(* CODESYS project tc3_hbi_mc2.library
   Company: BeckHoff
   DefaultNamespace: Tc3_HBI_MC2
   Version: 3.7.2.1
   Placeholder: Tc3_HBI_MC2
   Title: Tc3_HBI_MC2

Project tree, tasks and I/O mapping:
  libraries: Tc2_Drive, * (Beckhoff Automation GmbH); Tc2_EtherCAT, * (Beckhoff Automation GmbH); Tc2_MC2, * (Beckhoff Automation GmbH); Tc2_MC2_Drive, * (Beckhoff Automation GmbH); Tc2_Standard, * (Beckhoff Automation GmbH); Tc2_System, * (Beckhoff Automation GmbH); Tc2_Utilities, * (Beckhoff Automation GmbH); Tc3_HBI_System, * (BeckHoff); Tc3_Interfaces, * (Beckhoff Automation GmbH); Tc3_Module, * (Beckhoff Automation GmbH); Tc3_System, * (Beckhoff Automation GmbH)
  MOTION/
    POUs/
      FBs/
        [Internal]/
          DUTs/
            Basic/
              RegCorrection/
                data type _ST_MC2_RegCorrection_Get
                data type _ST_MC2_RegCorrection_Set
              data type _ST_MC2_AX5000_Status
              data type _ST_MC2_AX8000_Status
              data type _ST_MC2_Basic
              data type _ST_MC2_Basic_Status
              data type _ST_MC2_Dynamic
              data type _ST_MC2_EL70xx_Status
              data type _ST_MC2_EL72xx_Status
              data type _ST_MC2_Param1
              data type _ST_MC2_Param2
              data type _ST_MC2_SUB_Param
            Compact/
              data type _ST_MC2_Compact_Status
        Basic/
          DUTs/
            data type E_MC2_AX5000_Brake
            data type E_MC2_AX8000_Brake
            data type ST_MC2_AX5000
            data type ST_MC2_AX8000
            data type ST_MC2_Basic
            data type ST_MC2_EL70xx
            data type ST_MC2_EL72xx
            data type ST_MC2_RegCorrection
          ITFs/
            interface I_MC2_AX5000: M_nMC_AcceptBlockedDriveSignal, M_nMC_Brake, M_nMC_ClrLagError, M_nMC_MotorParam1, M_nMC_PID_PosCtrl, M_nMC_Power, M_nMC_Torque, M_nMC_TouchProbe1, M_nMC_TouchProbe2, M_nReset, P_lrRecordedPosition1_RisingEdge, P_lrRecordedPosition2_FallingEdge, P_lrRecordedPosition2_RisingEdge, P_nDiagnosticNumber, P_rActualMainVoltage, P_rAmplifierTemperature, P_rMotorTemperature, P_sDiagnosticNumber
            interface I_MC2_Basic: M_nMC_ClrLagError, M_nMC_DeadTimeComp, M_nMC_GearIn, M_nMC_GearInDyn, M_nMC_GearInMultiMaster, M_nMC_GearOut, M_nMC_InverseMotor, M_nMC_PhasingAbsolute, M_nMC_PhasingRelative, M_nMC_PositionLagMonitoring, M_nMC_Power, M_nMC_RegCorrection, M_nMC_SetEncoderOffset, M_nMC_SetFeedConstant, M_nMC_SetModuloFactor, M_nMC_SetPosition, M_nMC_SetPositionRelative, M_nMC_SetScaleFactor, M_nMC_SetVeloKvFactor, M_nReset, P_bAdvancedSlaveDynamics, P_bInGear, P_lrAbsolutePhaseShift, P_lrCoveredPhaseShift, P_lrGearRatio1, P_lrGearRatio2, P_lrGearRatio3, P_lrGearRatio4, P_lrMaxVelocity, P_lrModuloFactor
            interface I_MC2_EL70xx: P_rAmplifierTemperature, P_rControlVoltage, P_rMotorSupplyVoltage
            interface I_MC2_EL72xx: P_rAmplifierTemperature, P_rMotorSupplyVoltage, P_rMotorTemperature
          function block FB_MC2_AX5000 [ST]: M_nMC_AcceptBlockedDriveSignal, M_nMC_Brake, M_nMC_ClrLagError, M_nMC_DriveData, M_nMC_MotorParam1, M_nMC_PID_PosCtrl, M_nMC_Power, M_nMC_Torque, M_nMC_TouchProbe1, M_nMC_TouchProbe2, M_nReset, P_lrRecordedPosition1_RisingEdge, P_lrRecordedPosition2_FallingEdge, P_lrRecordedPosition2_RisingEdge, P_nDiagnosticNumber, P_rActualMainVoltage, P_rAmplifierTemperature, P_rMotorTemperature, P_sDiagnosticNumber
          function block FB_MC2_AX8000 [ST]: M_nMC_Brake, M_nMC_DriveData, M_nMC_Power, M_nMC_Torque, M_nReset, P_rActualMainVoltage, P_rAmplifierTemperature, P_rMotorTemperature
          function block FB_MC2_Basic [ST]: M_nMC_ClrLagError, M_nMC_DeadTimeComp, M_nMC_GearIn, M_nMC_GearInDyn, M_nMC_GearInMultiMaster, M_nMC_GearOut, M_nMC_InverseMotor, M_nMC_PhasingAbsolute, M_nMC_PhasingRelative, M_nMC_PositionLagMonitoring, M_nMC_Power, M_nMC_ReadParameter, M_nMC_RegCorrection, M_nMC_SetEncoderOffset, M_nMC_SetFeedConstant, M_nMC_SetModuloFactor, M_nMC_SetPosition, M_nMC_SetPositionRelative, M_nMC_SetScaleFactor, M_nMC_SetVeloKvFactor, M_nReset, P_bAdvancedSlaveDynamics, P_bInGear, P_lrAbsolutePhaseShift, P_lrCoveredPhaseShift, P_lrGearRatio1, P_lrGearRatio2, P_lrGearRatio3, P_lrGearRatio4, P_lrMaxVelocity, P_lrModuloFactor
          function block FB_MC2_EL70xx [ST]: M_nMC_DriveData, M_nMC_Power, P_rAmplifierTemperature, P_rControlVoltage, P_rMotorSupplyVoltage
          function block FB_MC2_EL72xx [ST]: M_nMC_DriveData, M_nMC_Power, P_rAmplifierTemperature, P_rMotorSupplyVoltage, P_rMotorTemperature
        Compact/
          DUTs/
            data type ST_MC2_Compact
          ITFs/
            interface I_MC2_Compact: M_nMC_Dynamic, M_nMC_Halt, M_nMC_Home, M_nMC_HomeReset, M_nMC_Jog, M_nMC_MoveAbsolute, M_nMC_MoveModulo, M_nMC_MoveRelative, M_nMC_MoveVelocity, M_nMC_Power, M_nMC_QuickStop, M_nMC_Stop, M_nReset, P_bE_Stop, P_bE_StopDelay, P_bEnable, P_bEnable_Negative, P_bEnable_Positive, P_bHardwareConnected, P_bHomed, P_eBufferMode, P_lrOverride, P_pAXIS_REF, P_pDriveAddress, P_stDynamic
          function block FB_MC2_Compact [ST]: M_nMC_Dynamic, M_nMC_Halt, M_nMC_Home, M_nMC_HomeReset, M_nMC_Jog, M_nMC_Local_Halt, M_nMC_MoveAbsolute, M_nMC_MoveModulo, M_nMC_MoveRelative, M_nMC_MoveVelocity, M_nMC_Power, M_nMC_QuickStop, M_nMC_ReadDriveAddress, M_nMC_Stop, M_nReset, P_bE_Stop, P_bE_StopDelay, P_bEnable, P_bEnable_Negative, P_bEnable_Positive, P_bHardwareConnected, P_bHomed, P_eBufferMode, P_lrOverride, P_pAXIS_REF, P_pDriveAddress, P_sMessage, P_stDynamic
          function block FB_MC2_Compact_AX8000 [ST]: M_nMC_DriveData, M_nMC_Power, M_nReset, P_rActualMainVoltage, P_rAmplifierTemperature, P_rMotorTemperature
  Version/
    global variables Global_Version
  Tc3_HBI_MC2.tmc
*)

// MOTION/POUs/FBs/[Internal]/DUTs/Basic/RegCorrection/_ST_MC2_RegCorrection_Get
{attribute 'hide'}
TYPE _ST_MC2_RegCorrection_Get :
STRUCT
	bWarning: BOOL; 
	nWarningId: UDINT; 
	lrActualVelocityDiff: LREAL; 
	lrActualDistance: LREAL; 
	lrActualLength: LREAL; 
	lrActualAcceleration: LREAL; 
	lrActualDeceleration: LREAL;
END_STRUCT
END_TYPE

// MOTION/POUs/FBs/[Internal]/DUTs/Basic/RegCorrection/_ST_MC2_RegCorrection_Set
{attribute 'hide'}
TYPE _ST_MC2_RegCorrection_Set :
STRUCT
	eMode: Tc2_MC2.E_SuperpositionMode:= Tc2_MC2.SUPERPOSITIONMODE_LENGTHREDUCTION_LIMITEDMOTION;
	lrDistance: LREAL:= 10.0; 
	lrVelocityDiff: LREAL:= 30.0; 
	lrAcceleration: LREAL:= 0.0; 
	lrDeceleration: LREAL:= 0.0; 
	lrJerk: LREAL:= 0.0; 
	lrVelocityProcess: LREAL:= 50.0; 
	lrLength: LREAL:= 360.0;
	eOptions: Tc2_MC2.ST_SuperpositionOptions;
END_STRUCT
END_TYPE

// MOTION/POUs/FBs/[Internal]/DUTs/Basic/_ST_MC2_AX5000_Status
TYPE _ST_MC2_AX5000_Status EXTENDS _ST_MC2_Basic_Status:
STRUCT
	nMC_AcceptBlockedDriveSignal: UDINT;	
	nMC_Brake: UDINT;
	nMC_FeedConstant: UDINT;
	nMC_MotorParam1: UDINT;
	nMC_PID_PosCtrl: UDINT;
	nMC_Torque: UDINT;
	nMC_TouchProbe1: UDINT;
	nMC_TouchProbe2: UDINT;
END_STRUCT
END_TYPE

// MOTION/POUs/FBs/[Internal]/DUTs/Basic/_ST_MC2_AX8000_Status
TYPE _ST_MC2_AX8000_Status EXTENDS _ST_MC2_Basic_Status :
STRUCT
	nMC_Brake: UDINT;	
	nMC_Torque: UDINT;
END_STRUCT
END_TYPE

// MOTION/POUs/FBs/[Internal]/DUTs/Basic/_ST_MC2_Basic
TYPE _ST_MC2_Basic EXTENDS Tc3_HBI_System.ST_Basic :
STRUCT
	bEnable: BOOL;
	bEnable_Negative: BOOL;
	bEnable_Positive: BOOL;
	lrOverride: LREAL;
	lrQuickStopRamp: LREAL;
	bE_Stop: BOOL;
	bE_StopDelay: BOOL;
	bExecute: BOOL;	
	bHome: BOOL;
	bResetHomed: BOOL;	
	bCalibrationCam	: BOOL;
	lrHomePosition	: LREAL;
	bHalt	: BOOL;
	bStop	: BOOL;
	bAbsMove	: BOOL;
	lrAbsPosition	: LREAL;
	lrAbsVelocity	: LREAL;
	bRelMove	: BOOL;
	lrRelDistance	: LREAL;
	lrRelVelocity	: LREAL;
	bMoveVelo	: BOOL;
	lrVeloVelocity	: LREAL;
	bJogForward: BOOL;
	bJogBackwards: BOOL;
	lrJogVelocity	: LREAL;
	lrAcceleration	: LREAL;
	lrDecelaration	: LREAL;
	lrJerk			: LREAL;
	bMoveModulo	: BOOL;
	lrModuloPosition	: LREAL;
	lrModuloVelocity	: LREAL;
	bSetDynamic	: BOOL;
	bReadDriveAddress	: BOOL;
	bPositiveLimit	: BOOL;							
	bNegativeLimit	: BOOL;	

	bSetEncoderOffset: BOOL;
	lrEncoderOffset: LREAL;
	bSetPosition: BOOL;
	lrSetPosotion	: LREAL;						
	
	eBufferMode	: Tc2_MC2.MC_BufferMode;
	eHomingMode	: Tc2_MC2.MC_HomingMode;
	eJogMode		: Tc2_MC2.E_JogMode;
	eDirection		: Tc2_MC2.MC_Direction;
	tHomeTimeout	: TIME;
	tMovementTimeout: TIME;

	bInGear: BOOL;
	lrGearRatio1: LREAL;
	lrGearRatio2: LREAL;
	lrGearRatio3: LREAL;
	lrGearRatio4: LREAL;
	lrModuloFactor: LREAL;
	lrMaxVelocity: LREAL;
	lrAbsolutePhaseShift: LREAL;
	lrCoveredPhaseShift: LREAL;
	stRegCorrection_Get: _ST_MC2_RegCorrection_Get;
END_STRUCT
END_TYPE

// MOTION/POUs/FBs/[Internal]/DUTs/Basic/_ST_MC2_Basic_Status
TYPE _ST_MC2_Basic_Status EXTENDS _ST_MC2_Compact_Status:
STRUCT
	nMC_ClrLagError: UDINT;
	nMC_DeadTimeComp: UDINT;
	nMC_GearIn: UDINT;
	nMC_GearInDyn: UDINT;
	nMC_GearInMultiMaster: UDINT;
	nMC_GearInMultiMaster_Dynamic : UDINT;
	nMC_GearOut: UDINT;
	nMC_InverseMotor: UDINT;
	nMC_PositionLagMonitoring: UDINT;
	nMC_RegCorrection: UDINT;
	nMC_SetFeedConstant: UDINT;
	nMC_SetEncoderOffset: UDINT;
	nMC_SetModuloFactor: UDINT;
	nMC_SetVeloKvFactor: UDINT;
	nMC_SetPosition: UDINT;
	nMC_SetPositionRelative: UDINT;
	nMC_SetScaleFactor: UDINT;
	nMC_PhasingAbsolute: UDINT;
	nMC_PhasingRelative: UDINT;
END_STRUCT
END_TYPE

// MOTION/POUs/FBs/[Internal]/DUTs/Basic/_ST_MC2_Dynamic
TYPE _ST_MC2_Dynamic :
STRUCT
	lrAcceleration: LREAL;
	lrDeceleration: LREAL;
	lrJerk: LREAL;
END_STRUCT
END_TYPE

// MOTION/POUs/FBs/[Internal]/DUTs/Basic/_ST_MC2_EL70xx_Status
TYPE _ST_MC2_EL70xx_Status EXTENDS _ST_MC2_Basic_Status:
STRUCT
END_STRUCT
END_TYPE

// MOTION/POUs/FBs/[Internal]/DUTs/Basic/_ST_MC2_EL72xx_Status
TYPE _ST_MC2_EL72xx_Status EXTENDS _ST_MC2_Basic_Status:
STRUCT
END_STRUCT
END_TYPE

// MOTION/POUs/FBs/[Internal]/DUTs/Basic/_ST_MC2_Param1
{attribute 'hide'}
TYPE _ST_MC2_Param1 :
STRUCT
	aParm: ARRAY[1..6] OF _ST_MC2_SUB_Param;
	nEncoderDir: WORD;
	nMotorDir: WORD;
	nHomeCamDir: WORD;
	nHomeSyncDir: WORD;
	lrRefVelocity: LREAL;
	lrMaxVelocity: LREAL;
END_STRUCT
END_TYPE

// MOTION/POUs/FBs/[Internal]/DUTs/Basic/_ST_MC2_Param2
{attribute 'hide'}
TYPE _ST_MC2_Param2 :
STRUCT
	aParm: ARRAY[1..4] OF _ST_MC2_SUB_Param;
	nEncoderDir: WORD;
	nMotorDir: WORD;
	nHomeCamDir: WORD;
	nHomeSyncDir: WORD;
END_STRUCT
END_TYPE

// MOTION/POUs/FBs/[Internal]/DUTs/Basic/_ST_MC2_SUB_Param
{attribute 'hide'}
TYPE _ST_MC2_SUB_Param :
STRUCT
	nIndexGroup: UDINT;
	nIndexOffset: UDINT;
	nDataSize: UDINT;
END_STRUCT
END_TYPE

// MOTION/POUs/FBs/[Internal]/DUTs/Compact/_ST_MC2_Compact_Status
TYPE _ST_MC2_Compact_Status:
STRUCT
	bHomed: BOOL;
	lrActPos: LREAL;
	lrActVelocity: LREAL;
	nMC_Dynamic: UDINT;
	nMC_Halt: UDINT;
	nMC_Home: UDINT;
	nMC_HomeReset: UDINT;
	nMC_Jog: UDINT;
	M_nMC_Local_Halt: UDINT;
	nMC_MoveAbsolute: UDINT;
	nMC_MoveModulo: UDINT;
	nMC_MoveRelative: UDINT;
	nMC_MoveVelocity: UDINT;
	nMC_Power: UDINT;
	nMC_QuickStop: UDINT;
	M_nMC_ReadDriveAddress: UDINT;
	nMC_Stop: UDINT;
	nReset: UDINT;
END_STRUCT
END_TYPE

// MOTION/POUs/FBs/Basic/DUTs/E_MC2_AX5000_Brake
TYPE E_MC2_AX5000_Brake :
(
	AX5000_Brake_Automatic,	
	AX5000_Brake_Force_lock,	
	AX5000_Brake_Force_unlock
);
END_TYPE

// MOTION/POUs/FBs/Basic/DUTs/E_MC2_AX8000_Brake
TYPE E_MC2_AX8000_Brake :
(
	AX8000_Brake_Release_force,	
	AX8000_Brake_Force_lock,	
	AX8000_Brake_Force_unlock
);
END_TYPE

// MOTION/POUs/FBs/Basic/DUTs/ST_MC2_AX5000
TYPE ST_MC2_AX5000 EXTENDS _ST_MC2_Basic :
STRUCT
	lrRecordedPosition1_RisingEdge: LREAL;
	lrRecordedPosition2_RisingEdge: LREAL;	
	lrRecordedPosition2_FallingEdge: LREAL;		
	rActualMainVoltage: REAL;
	rAmplifierTemperature: REAL;
	rMotorTemperature: REAL;
	nDiagnosticNumber: UDINT;
	sDiagnosticNumber: STRING;
	stStatus: _ST_MC2_AX5000_Status;
END_STRUCT
END_TYPE

// MOTION/POUs/FBs/Basic/DUTs/ST_MC2_AX8000
TYPE ST_MC2_AX8000 EXTENDS _ST_MC2_Basic :
STRUCT
	rActualMainVoltage: REAL;
	rAmplifierTemperature: REAL;
	rMotorTemperature: REAL;
	stStatus: _ST_MC2_AX8000_Status;
END_STRUCT
END_TYPE

// MOTION/POUs/FBs/Basic/DUTs/ST_MC2_Basic
TYPE ST_MC2_Basic EXTENDS _ST_MC2_Basic :
STRUCT
	stStatus: _ST_MC2_Basic_Status;
END_STRUCT
END_TYPE

// MOTION/POUs/FBs/Basic/DUTs/ST_MC2_EL70xx
TYPE ST_MC2_EL70xx EXTENDS _ST_MC2_Basic :
STRUCT
	rAmplifierTemperature: REAL;
	rControlVoltage: REAL;
	rMotorSupplyVoltage: REAL;
	stStatus: _ST_MC2_EL70xx_Status;
END_STRUCT
END_TYPE

// MOTION/POUs/FBs/Basic/DUTs/ST_MC2_EL72xx
TYPE ST_MC2_EL72xx EXTENDS _ST_MC2_Basic :
STRUCT
	rAmplifierTemperature: REAL;
	rMotorSupplyVoltage: REAL;
	rMotorTemperature: REAL;
	stStatus: _ST_MC2_EL72xx_Status;
END_STRUCT
END_TYPE

// MOTION/POUs/FBs/Basic/DUTs/ST_MC2_RegCorrection
TYPE ST_MC2_RegCorrection :
STRUCT
	Set: _ST_MC2_RegCorrection_Set;
	Get: _ST_MC2_RegCorrection_Get;  	
END_STRUCT
END_TYPE

// MOTION/POUs/FBs/Compact/DUTs/ST_MC2_Compact
TYPE ST_MC2_Compact EXTENDS ST_Basic :
STRUCT
	bEnable: BOOL;
	bEnable_Negative: BOOL;
	bEnable_Positive: BOOL;
	lrOverride: LREAL;
	lrQuickStopRamp: LREAL;
	bE_Stop: BOOL;
	bE_StopDelay: BOOL;
	bExecute: BOOL;	
	bHome: BOOL;
	bResetHomed: BOOL;	
	bCalibrationCam	: BOOL;
	lrHomePosition	: LREAL;
	bHalt	: BOOL;
	bStop	: BOOL;
	bAbsMove	: BOOL;
	lrAbsPosition	: LREAL;
	lrAbsVelocity	: LREAL;
	bRelMove	: BOOL;
	lrRelDistance	: LREAL;
	lrRelVelocity	: LREAL;
	bMoveVelo	: BOOL;
	lrVeloVelocity	: LREAL;
	bJogForward: BOOL;
	bJogBackwards: BOOL;
	lrJogVelocity	: LREAL;
	lrAcceleration	: LREAL;
	lrDecelaration	: LREAL;
	lrJerk			: LREAL;
	bMoveModulo	: BOOL;
	lrModuloPosition	: LREAL;
	lrModuloVelocity	: LREAL;
	bSetDynamic	: BOOL;
	bReadDriveAddress	: BOOL;
	bPositiveLimit	: BOOL;							
	bNegativeLimit	: BOOL;							
	eBufferMode	: Tc2_MC2.MC_BufferMode;
	eHomingMode	: Tc2_MC2.MC_HomingMode;
	eJogMode		: Tc2_MC2.E_JogMode;
	eDirection		: Tc2_MC2.MC_Direction;
	tHomeTimeout	: TIME;
	tMovementTimeout: TIME;
	stStatus: _ST_MC2_Compact_Status;
END_STRUCT
END_TYPE

// Version/Global_Version
{attribute 'TcGenerated'}
// This function has been automatically generated from the project information.
VAR_GLOBAL CONSTANT
	{attribute 'const_non_replaced'}
	{attribute 'linkalways'}
	stLibVersion_Tc3_HBI_MC2 : ST_LibVersion := (iMajor := 3, iMinor := 7, iBuild := 2, iRevision := 1, sVersion := '3.7.2.1');
END_VAR

// MOTION/POUs/FBs/Basic/ITFs/I_MC2_AX5000
INTERFACE I_MC2_AX5000 EXTENDS I_MC2_Basic

//	The result of the method is an unsigned double integer
//	0 = idle 
//	1 = coupled
//	2 = starting
//	3 = running
//	4 = aborted
// 	5 = no hardware connected
// 	6 = Spare
//	7 = pointer or index error
//	8 = mapping error
//	9 = parameter error
//	10 = complete
//	Any other number = ErrorID
METHOD PUBLIC M_nMC_AcceptBlockedDriveSignal : UDINT
VAR_INPUT
	bExecute: BOOL;
END_VAR
END_METHOD

//	The result of the method is an unsigned double integer
//	0 = idle 
//	1 = coupled
//	2 = starting
//	3 = running
//	4 = aborted
// 	5 = no hardware connected
// 	6 = Spare
//	7 = pointer or index error
//	8 = mapping error
//	9 = parameter error
//	10 = complete
//	Any other number = ErrorID
METHOD PUBLIC M_nMC_Brake : UDINT
VAR_INPUT
	bExecute: BOOL;
	eBrakeState: E_MC2_AX5000_Brake;
END_VAR
END_METHOD

//	The result of the method is an unsigned double integer
//	0 = idle 
//	1 = coupled
//	2 = starting
//	3 = running
//	4 = aborted
// 	5 = no hardware connected
// 	6 = Spare
//	7 = pointer or index error
//	8 = mapping error
//	9 = parameter error
//	10 = complete
//	Any other number = ErrorID
METHOD PUBLIC M_nMC_ClrLagError : UDINT
VAR_INPUT
	bExecute: BOOL;
END_VAR
END_METHOD

//	The result of the method is an unsigned double integer
//	0 = idle 
//	1 = coupled
//	2 = starting
//	3 = running
//	4 = aborted
// 	5 = no hardware connected
// 	6 = Spare
//	7 = pointer or index error
//	8 = mapping error
//	9 = parameter error
//	10 = complete
//	Any other number = ErrorID
METHOD PUBLIC M_nMC_MotorParam1 : UDINT
VAR_INPUT
	bExecute: BOOL;
	bInverse: BOOL;
	nMaxRpm: UINT;
	lrDiameter: LREAL;
	lrGearNumerator: LREAL;
	lrGearDenominator: LREAL;
END_VAR
END_METHOD

//	The result of the method is an unsigned double integer
//	0 = idle 
//	1 = coupled
//	2 = starting
//	3 = running
//	4 = aborted
// 	5 = no hardware connected
// 	6 = Spare
//	7 = pointer or index error
//	8 = mapping error
//	9 = parameter error
//	10 = complete
//	Any other number = ErrorID
METHOD PUBLIC M_nMC_PID_PosCtrl : UDINT
VAR_INPUT
	bExecute: BOOL;
	rKv: REAL; 		// 0.0 - 100.0 
END_VAR
END_METHOD

//	The result of the method is an unsigned double integer
//	0 = idle 
//	1 = coupled
//	2 = starting
//	3 = running
//	4 = aborted
// 	5 = no hardware connected
// 	6 = Spare
//	7 = pointer or index error
//	8 = mapping error
//	9 = parameter error
//	10 = complete
//	Any other number = ErrorID
METHOD PUBLIC M_nMC_Power : UDINT
VAR_INPUT
	bEnable: BOOL;
	bE_Stop: BOOL;
	bE_StopDelay: BOOL;
	bEnable_Positive: BOOL;
	bEnable_Negative: BOOL;
END_VAR
END_METHOD

//	The result of the method is an unsigned double integer
//	0 = idle 
//	1 = coupled
//	2 = starting
//	3 = running
//	4 = aborted
// 	5 = no hardware connected
// 	6 = Spare
//	7 = pointer or index error
//	8 = mapping error
//	9 = parameter error
//	10 = complete
//	Any other number = ErrorID
METHOD PUBLIC M_nMC_Torque : UDINT
VAR_INPUT
	bExecute: BOOL;
	lrTorque: LREAL; 		// Torque limit 0.0-100.0%	
END_VAR
END_METHOD

//	The result of the method is an unsigned double integer
//	0 = idle 
//	1 = coupled
//	2 = starting
//	3 = running
//	4 = aborted
// 	5 = no hardware connected
// 	6 = Spare
//	7 = pointer or index error
//	8 = mapping error
//	9 = parameter error
//	10 = complete
//	Any other number = ErrorID
METHOD PUBLIC M_nMC_TouchProbe1 : UDINT
VAR_INPUT
	bEnable: BOOL;
	lrPrellFilter_RisingEdge: LREAL;
END_VAR
END_METHOD

//	The result of the method is an unsigned double integer
//	0 = idle 
//	1 = coupled
//	2 = starting
//	3 = running
//	4 = aborted
// 	5 = no hardware connected
// 	6 = Spare
//	7 = pointer or index error
//	8 = mapping error
//	9 = parameter error
//	10 = complete
//	Any other number = ErrorID
METHOD PUBLIC M_nMC_TouchProbe2 : UDINT
VAR_INPUT
	bEnable: BOOL;
	lrPrellFilter_RisingEdge: LREAL;
	lrPrellFilter_FallingEdge: LREAL;
END_VAR
END_METHOD

//	The result of the method is an unsigned double integer
//	0 = idle 
//	1 = coupled
//	2 = starting
//	3 = running
//	4 = aborted
// 	5 = no hardware connected
// 	6 = Spare
//	7 = pointer or index error
//	8 = mapping error
//	9 = parameter error
//	10 = complete
//	Any other number = ErrorID
METHOD PUBLIC M_nReset : UDINT
VAR_INPUT
	bExecute: BOOL;
END_VAR
END_METHOD

PROPERTY PUBLIC P_lrRecordedPosition1_RisingEdge : LREAL
GET
END_GET
END_PROPERTY

PROPERTY PUBLIC P_lrRecordedPosition2_FallingEdge : LREAL
GET
END_GET
END_PROPERTY

PROPERTY PUBLIC P_lrRecordedPosition2_RisingEdge : LREAL
GET
END_GET
END_PROPERTY

PROPERTY PUBLIC P_nDiagnosticNumber : UDINT
GET
END_GET
END_PROPERTY

PROPERTY PUBLIC P_rActualMainVoltage : REAL
GET
END_GET
END_PROPERTY

PROPERTY PUBLIC P_rAmplifierTemperature : REAL
GET
END_GET
END_PROPERTY

PROPERTY PUBLIC P_rMotorTemperature : REAL
GET
END_GET
END_PROPERTY

PROPERTY PUBLIC P_sDiagnosticNumber : STRING
GET
END_GET
END_PROPERTY

END_INTERFACE

// MOTION/POUs/FBs/Basic/ITFs/I_MC2_Basic
INTERFACE I_MC2_Basic EXTENDS I_MC2_Compact

//	The result of the method is an unsigned double integer
//	0 = idle 
//	1 = coupled
//	2 = starting
//	3 = running
//	4 = aborted
// 	5 = no hardware connected
// 	6 = Spare
//	7 = pointer or index error
//	8 = mapping error
//	9 = parameter error
//	10 = complete
//	Any other number = ErrorID
METHOD PUBLIC M_nMC_ClrLagError : UDINT
VAR_INPUT
	bExecute: BOOL;
END_VAR
END_METHOD

//	The result of the method is an unsigned double integer
//	0 = idle 
//	1 = coupled
//	2 = starting
//	3 = running
//	4 = aborted
// 	5 = no hardware connected
// 	6 = Spare
//	7 = pointer or index error
//	8 = mapping error
//	9 = parameter error
//	10 = complete
//	Any other number = ErrorID
METHOD PUBLIC M_nMC_DeadTimeComp : UDINT
END_METHOD

//	The result of the method is an unsigned double integer
//	0 = idle 
//	1 = coupled
//	2 = starting
//	3 = running
//	4 = aborted
// 	5 = no hardware connected
// 	6 = Spare
//	7 = pointer or index error
//	8 = mapping error
//	9 = parameter error
//	10 = complete
//	Any other number = ErrorID
METHOD PUBLIC M_nMC_GearIn : UDINT
VAR_INPUT
	bExecute: BOOL;
	pMaster: POINTER TO TC2_MC2.AXIS_REF;
	lrRatioNumerator: LREAL;
	iRatioDenominator: UINT;
END_VAR
END_METHOD

//	The result of the method is an unsigned double integer
//	0 = idle 
//	1 = coupled
//	2 = starting
//	3 = running
//	4 = aborted
// 	5 = no hardware
//	7 = pointer or index error
//	8 = mapping error
//	9 = parameter error
//	10 = complete
//	Any other number = ErrorID
METHOD PUBLIC M_nMC_GearInDyn : UDINT
VAR_INPUT
	bEnable: BOOL;
	pMaster: POINTER TO TC2_MC2.AXIS_REF;
	lrGearRatio: LREAL;
END_VAR
END_METHOD

//	The result of the method is an unsigned double integer
//	0 = idle 
//	1 = coupled
//	2 = starting
//	3 = running
//	4 = aborted
// 	5 = no hardware connected
// 	6 = Spare
//	7 = pointer or index error
//	8 = mapping error
//	9 = parameter error
//	10 = complete
//	Any other number = ErrorID
METHOD PUBLIC M_nMC_GearInMultiMaster : UDINT
VAR_INPUT
	bEnable: BOOL;
	pMaster1: POINTER TO Tc2_MC2.AXIS_REF;
	pMaster2: POINTER TO Tc2_MC2.AXIS_REF;
	pMaster3: POINTER TO Tc2_MC2.AXIS_REF;
	pMaster4: POINTER TO Tc2_MC2.AXIS_REF;
END_VAR
END_METHOD

//	The result of the method is an unsigned double integer
//	0 = idle 
//	1 = coupled
//	2 = starting
//	3 = running
//	4 = aborted
// 	5 = no hardware connected
// 	6 = Spare
//	7 = pointer or index error
//	8 = mapping error
//	9 = parameter error
//	10 = complete
//	Any other number = ErrorID
METHOD PUBLIC M_nMC_GearOut : UDINT
VAR_INPUT
	bExecute: BOOL;
END_VAR
END_METHOD

//	The result of the method is an unsigned double integer
//	0 = idle 
//	1 = coupled
//	2 = starting
//	3 = running
//	4 = aborted
// 	5 = no hardware connected
// 	6 = Spare
//	7 = pointer or index error
//	8 = mapping error
//	9 = parameter error
//	10 = complete
//	Any other number = ErrorID
METHOD PUBLIC M_nMC_InverseMotor : UDINT
VAR_INPUT
	bExecute: BOOL;
	bInverse: BOOL;
END_VAR
END_METHOD

//	The result of the method is an unsigned double integer
//	0 = idle 
//	1 = coupled
//	2 = starting
//	3 = running
//	4 = aborted
// 	5 = no hardware connected
// 	6 = Spare
//	7 = pointer or index error
//	8 = mapping error
//	9 = parameter error
//	10 = complete
//	Any other number = ErrorID
METHOD PUBLIC M_nMC_PhasingAbsolute : UDINT
VAR_INPUT
	bExecute: BOOL;
	pMaster: POINTER TO TC2_MC2.AXIS_REF;
	lrPhaseShift: LREAL;
	lrVelocity: LREAL;
END_VAR
END_METHOD

//	The result of the method is an unsigned double integer
//	0 = idle 
//	1 = coupled
//	2 = starting
//	3 = running
//	4 = aborted
// 	5 = no hardware connected
// 	6 = Spare
//	7 = pointer or index error
//	8 = mapping error
//	9 = parameter error
//	10 = complete
//	Any other number = ErrorID
METHOD PUBLIC M_nMC_PhasingRelative : UDINT
VAR_INPUT
	bExecute: BOOL;
	pMaster: POINTER TO TC2_MC2.AXIS_REF;
	lrPhaseShift: LREAL;
	lrVelocity: LREAL;
END_VAR
END_METHOD

//	The result of the method is an unsigned double integer
//	0 = idle 
//	1 = coupled
//	2 = starting
//	3 = running
//	4 = aborted
// 	5 = no hardware connected
// 	6 = Spare
//	7 = pointer or index error
//	8 = mapping error
//	9 = parameter error
//	10 = complete
//	Any other number = ErrorID
METHOD PUBLIC M_nMC_PositionLagMonitoring : UDINT
VAR_INPUT
	bEnable: BOOL;
	bDisable: BOOL;
END_VAR
END_METHOD

//	The result of the method is an unsigned double integer
//	0 = idle 
//	1 = coupled
//	2 = starting
//	3 = running
//	4 = aborted
// 	5 = no hardware connected
// 	6 = Spare
//	7 = pointer or index error
//	8 = mapping error
//	9 = parameter error
//	10 = complete
//	Any other number = ErrorID
METHOD PUBLIC M_nMC_Power : UDINT
VAR_INPUT
	bEnable: BOOL;
	bE_Stop: BOOL;
	bE_StopDelay: BOOL;
	bEnable_Positive: BOOL;
	bEnable_Negative: BOOL;
END_VAR
END_METHOD

//	The result of the method is an unsigned double integer
//	0 = idle 
//	1 = coupled
//	2 = starting
//	3 = running
//	4 = aborted
// 	5 = no hardware connected
// 	6 = Spare
//	7 = pointer or index error
//	8 = mapping error
//	9 = parameter error
//	10 = complete
//	Any other number = ErrorID
METHOD PUBLIC M_nMC_RegCorrection : UDINT
VAR_INPUT
	bExecute: BOOL;
	pRegCorrection: POINTER TO ST_MC2_RegCorrection;
END_VAR
END_METHOD

//	The result of the method is an unsigned double integer
//	0 = idle 
//	1 = coupled
//	2 = starting
//	3 = running
//	4 = aborted
// 	5 = no hardware connected
// 	6 = Spare
//	7 = pointer or index error
//	8 = mapping error
//	9 = parameter error
//	10 = complete
//	Any other number = ErrorID
METHOD PUBLIC M_nMC_SetEncoderOffset : UDINT
VAR_INPUT
	bExecute: BOOL;
	lrOffset: LREAL;
END_VAR
END_METHOD

//	The result of the method is an unsigned double integer
//	0 = idle 
//	1 = coupled
//	2 = starting
//	3 = running
//	4 = aborted
// 	5 = no hardware connected
// 	6 = Spare
//	7 = pointer or index error
//	8 = mapping error
//	9 = parameter error
//	10 = complete
//	Any other number = ErrorID
METHOD PUBLIC M_nMC_SetFeedConstant : UDINT
VAR_INPUT
	bExecute: BOOL;
	lrFeedConstant: LREAL;
END_VAR
END_METHOD

//	The result of the method is an unsigned double integer
//	0 = idle 
//	1 = coupled
//	2 = starting
//	3 = running
//	4 = aborted
// 	5 = no hardware connected
// 	6 = Spare
//	7 = pointer or index error
//	8 = mapping error
//	9 = parameter error
//	10 = complete
//	Any other number = ErrorID
METHOD PUBLIC M_nMC_SetModuloFactor : UDINT
VAR_INPUT
	bExecute: BOOL;
	lrModuloFactor: LREAL;
END_VAR
END_METHOD

//	The result of the method is an unsigned double integer
//	0 = idle 
//	1 = coupled
//	2 = starting
//	3 = running
//	4 = aborted
// 	5 = no hardware connected
// 	6 = Spare
//	7 = pointer or index error
//	8 = mapping error
//	9 = parameter error
//	10 = complete
//	Any other number = ErrorID
METHOD PUBLIC M_nMC_SetPosition : UDINT
VAR_INPUT
	bExecute: BOOL;
	lrPosition: LREAL;
END_VAR
END_METHOD

//	The result of the method is an unsigned double integer
//	0 = idle 
//	1 = coupled
//	2 = starting
//	3 = running
//	4 = aborted
// 	5 = no hardware connected
// 	6 = Spare
//	7 = pointer or index error
//	8 = mapping error
//	9 = parameter error
//	10 = complete
//	Any other number = ErrorID
METHOD PUBLIC M_nMC_SetPositionRelative : UDINT
VAR_INPUT
	bExecute: BOOL;
	lrPosition: LREAL;
END_VAR
END_METHOD

//	The result of the method is an unsigned double integer
//	0 = idle 
//	1 = coupled
//	2 = starting
//	3 = running
//	4 = aborted
// 	5 = no hardware connected
// 	6 = Spare
//	7 = pointer or index error
//	8 = mapping error
//	9 = parameter error
//	10 = complete
//	Any other number = ErrorID
METHOD PUBLIC M_nMC_SetScaleFactor : UDINT
VAR_INPUT
	bExecute: BOOL;
	lrScaleFactor: LREAL;
END_VAR
END_METHOD

//	The result of the method is an unsigned double integer
//	0 = idle 
//	1 = coupled
//	2 = starting
//	3 = running
//	4 = aborted
// 	5 = no hardware connected
// 	6 = Spare
//	7 = pointer or index error
//	8 = mapping error
//	9 = parameter error
//	10 = complete
//	Any other number = ErrorID
METHOD PUBLIC M_nMC_SetVeloKvFactor : UDINT
VAR_INPUT
	bExecute: BOOL;
	lrKvFactor: LREAL;
END_VAR
END_METHOD

//	The result of the method is an unsigned double integer
//	0 = idle 
//	1 = coupled
//	2 = starting
//	3 = running
//	4 = aborted
// 	5 = no hardware connected
// 	6 = Spare
//	7 = pointer or index error
//	8 = mapping error
//	9 = parameter error
//	10 = complete
//	Any other number = ErrorID
METHOD PUBLIC M_nReset : UDINT
VAR_INPUT
	bExecute: BOOL;
END_VAR
END_METHOD

PROPERTY PUBLIC P_bAdvancedSlaveDynamics : BOOL
SET
END_SET
END_PROPERTY

PROPERTY PUBLIC P_bInGear : BOOL
GET
END_GET
END_PROPERTY

PROPERTY PUBLIC P_lrAbsolutePhaseShift  : lreal
GET
END_GET
END_PROPERTY

PROPERTY PUBLIC P_lrCoveredPhaseShift : lreal
GET
END_GET
END_PROPERTY

PROPERTY PUBLIC P_lrGearRatio1 : LREAL
SET
END_SET
END_PROPERTY

PROPERTY PUBLIC P_lrGearRatio2 : LREAL
SET
END_SET
END_PROPERTY

PROPERTY PUBLIC P_lrGearRatio3 : LREAL
SET
END_SET
END_PROPERTY

PROPERTY PUBLIC P_lrGearRatio4 : LREAL
SET
END_SET
END_PROPERTY

PROPERTY PUBLIC P_lrMaxVelocity : LREAL
GET
END_GET
END_PROPERTY

PROPERTY PUBLIC P_lrModuloFactor : LREAL
GET
END_GET
END_PROPERTY

END_INTERFACE

// MOTION/POUs/FBs/Compact/ITFs/I_MC2_Compact
INTERFACE I_MC2_Compact EXTENDS Tc3_HBI_System.I_Basic

//	The result of the method is an unsigned double integer
//	0 = idle 
//	1 = coupled
//	2 = starting
//	3 = running
//	4 = aborted
// 	5 = no hardware connected
// 	6 = Spare
//	7 = pointer or index error
//	8 = mapping error
//	9 = parameter error
//	10 = complete
//	Any other number = ErrorID
METHOD PUBLIC M_nMC_Dynamic : UDINT
VAR_INPUT
	bExecute: BOOL;
	lrAcceleration: LREAL;
	lrDeceleration: LREAL;
	lrJerk: LREAL;
END_VAR
END_METHOD

//	The result of the method is an unsigned double integer
//	0 = idle 
//	1 = coupled
//	2 = starting
//	3 = running
//	4 = aborted
// 	5 = no hardware connected
// 	6 = Spare
//	7 = pointer or index error
//	8 = mapping error
//	9 = parameter error
//	10 = complete
//	Any other number = ErrorID
METHOD PUBLIC M_nMC_Halt : UDINT
VAR_INPUT
	bExecute: BOOL;
END_VAR
END_METHOD

//	The result of the method is an unsigned double integer
//	0 = idle 
//	1 = coupled
//	2 = starting
//	3 = running
//	4 = aborted
// 	5 = no hardware connected
// 	6 = Spare
//	7 = pointer or index error
//	8 = mapping error
//	9 = parameter error
//	10 = complete
//	Any other number = ErrorID
METHOD PUBLIC M_nMC_Home : UDINT
VAR_INPUT
	bExecute: BOOL;
	lrPosition: LREAL;
	bCalibrationCam: BOOL;
	eHomingMode: MC_HomingMode;
END_VAR
END_METHOD

//	The result of the method is an unsigned double integer
//	0 = idle 
//	1 = coupled
//	2 = starting
//	3 = running
//	4 = aborted
// 	5 = no hardware connected
// 	6 = Spare
//	7 = pointer or index error
//	8 = mapping error
//	9 = parameter error
//	10 = complete
//	Any other number = ErrorID
METHOD PUBLIC M_nMC_HomeReset : UDINT
VAR_INPUT
	bExecute: BOOL;
END_VAR
END_METHOD

//	The result of the method is an unsigned double integer
//	0 = idle 
//	1 = coupled
//	2 = starting
//	3 = running
//	4 = aborted
// 	5 = no hardware connected
// 	6 = Spare
//	7 = pointer or index error
//	8 = mapping error
//	9 = parameter error
//	10 = complete
//	Any other number = ErrorID
METHOD PUBLIC M_nMC_Jog : UDINT
VAR_INPUT
	bForward: BOOL;
	bBackwards: BOOL;
	lrVelocity: LREAL;
END_VAR
END_METHOD

//	The result of the method is an unsigned double integer
//	0 = idle 
//	1 = coupled
//	2 = starting
//	3 = running
//	4 = aborted
// 	5 = no hardware connected
// 	6 = Spare
//	7 = pointer or index error
//	8 = mapping error
//	9 = parameter error
//	10 = complete
//	Any other number = ErrorID
METHOD PUBLIC M_nMC_MoveAbsolute : UDINT
VAR_INPUT
	bExecute: BOOL;
	lrPosition: LREAL;
	lrVelocity: LREAL;
END_VAR
END_METHOD

//	The result of the method is an unsigned double integer
//	0 = idle 
//	1 = coupled
//	2 = starting
//	3 = running
//	4 = aborted
// 	5 = no hardware connected
// 	6 = Spare
//	7 = pointer or index error
//	8 = mapping error
//	9 = parameter error
//	10 = complete
//	Any other number = ErrorID
METHOD PUBLIC M_nMC_MoveModulo : UDINT
VAR_INPUT
	bExecute: BOOL;
	lrPosition: LREAL;
	lrVelocity: LREAL;
	eDirection: Tc2_MC2.MC_Direction;
END_VAR
END_METHOD

//	The result of the method is an unsigned double integer
//	0 = idle 
//	1 = coupled
//	2 = starting
//	3 = running
//	4 = aborted
// 	5 = no hardware connected
// 	6 = Spare
//	7 = pointer or index error
//	8 = mapping error
//	9 = parameter error
//	10 = complete
//	Any other number = ErrorID
METHOD PUBLIC M_nMC_MoveRelative : UDINT
VAR_INPUT
	bExecute: BOOL;
	lrDistance: LREAL;
	lrVelocity: LREAL;
END_VAR
END_METHOD

//	The result of the method is an unsigned double integer
//	0 = idle 
//	1 = coupled
//	2 = starting
//	3 = running
//	4 = aborted
// 	5 = no hardware connected
// 	6 = Spare
//	7 = pointer or index error
//	8 = mapping error
//	9 = parameter error
//	10 = complete
//	Any other number = ErrorID
METHOD PUBLIC M_nMC_MoveVelocity : UDINT
VAR_INPUT
	bExecute: BOOL;
	lrVelocity: LREAL;
	eDirection: MC_Direction;
END_VAR
END_METHOD

//	The result of the method is an unsigned double integer
//	0 = idle 
//	1 = coupled
//	2 = starting
//	3 = running
//	4 = aborted
// 	5 = no hardware connected
// 	6 = Spare
//	7 = pointer or index error
//	8 = mapping error
//	9 = parameter error
//	10 = complete
//	Any other number = ErrorID
METHOD PUBLIC M_nMC_Power : UDINT
VAR_INPUT
	bEnable: BOOL;
	bE_Stop: BOOL;
	bE_StopDelay: BOOL;
	bEnable_Positive: BOOL;
	bEnable_Negative: BOOL;
END_VAR
END_METHOD

//	The result of the method is an unsigned double integer
//	0 = idle 
//	1 = coupled
//	2 = starting
//	3 = running
//	4 = aborted
// 	5 = no hardware connected
// 	6 = Spare
//	7 = pointer or index error
//	8 = mapping error
//	9 = parameter error
//	10 = complete
//	Any other number = ErrorID
METHOD PUBLIC M_nMC_QuickStop : UDINT
VAR_INPUT
	bExecute: BOOL;
	lrDeceleration: LREAL;
	lrJerk: LREAL;
END_VAR
END_METHOD

//	The result of the method is an unsigned double integer
//	0 = idle 
//	1 = coupled
//	2 = starting
//	3 = running
//	4 = aborted
// 	5 = no hardware connected
// 	6 = Spare
//	7 = pointer or index error
//	8 = mapping error
//	9 = parameter error
//	10 = complete
//	Any other number = ErrorID
METHOD PUBLIC M_nMC_Stop : UDINT
VAR_INPUT
	bExecute: BOOL;
END_VAR
END_METHOD

//	The result of the method is an unsigned double integer
//	0 = idle 
//	1 = coupled
//	2 = starting
//	3 = running
//	4 = aborted
// 	5 = no hardware connected
// 	6 = Spare
//	7 = pointer or index error
//	8 = mapping error
//	9 = parameter error
//	10 = complete
//	Any other number = ErrorID
METHOD PUBLIC M_nReset : UDINT
VAR_INPUT
	bExecute: BOOL;
END_VAR
END_METHOD

PROPERTY PUBLIC P_bE_Stop : BOOL
GET
END_GET
END_PROPERTY

PROPERTY PUBLIC P_bE_StopDelay : BOOL
GET
END_GET
END_PROPERTY

PROPERTY PUBLIC P_bEnable : BOOL
GET
END_GET
END_PROPERTY

PROPERTY PUBLIC P_bEnable_Negative : BOOL
GET
END_GET
END_PROPERTY

PROPERTY PUBLIC P_bEnable_Positive : BOOL
GET
END_GET
END_PROPERTY

PROPERTY PUBLIC P_bHardwareConnected : BOOL
GET
END_GET
END_PROPERTY

PROPERTY PUBLIC P_bHomed : BOOL
GET
END_GET
END_PROPERTY

PROPERTY PUBLIC P_eBufferMode : MC_BufferMode
SET
END_SET
END_PROPERTY

PROPERTY PUBLIC P_lrOverride : LREAL
GET
END_GET
SET
END_SET
END_PROPERTY

PROPERTY PUBLIC P_pAXIS_REF : POINTER TO AXIS_REF
GET
END_GET
END_PROPERTY

PROPERTY PUBLIC P_pDriveAddress : POINTER TO ST_AdsAddress
GET
END_GET
END_PROPERTY

PROPERTY PUBLIC P_stDynamic : _ST_MC2_Dynamic
GET
END_GET
END_PROPERTY

END_INTERFACE

// MOTION/POUs/FBs/Basic/ITFs/I_MC2_EL70xx
INTERFACE I_MC2_EL70xx EXTENDS I_MC2_Basic

PROPERTY PUBLIC P_rAmplifierTemperature : REAL
GET
END_GET
END_PROPERTY

PROPERTY PUBLIC P_rControlVoltage : REAL
GET
END_GET
END_PROPERTY

PROPERTY PUBLIC P_rMotorSupplyVoltage : REAL
GET
END_GET
END_PROPERTY

END_INTERFACE

// MOTION/POUs/FBs/Basic/ITFs/I_MC2_EL72xx
INTERFACE I_MC2_EL72xx EXTENDS I_MC2_Basic

PROPERTY PUBLIC P_rAmplifierTemperature : REAL
GET
END_GET
END_PROPERTY

PROPERTY PUBLIC P_rMotorSupplyVoltage : REAL
GET
END_GET
END_PROPERTY

PROPERTY PUBLIC P_rMotorTemperature : REAL
GET
END_GET
END_PROPERTY

END_INTERFACE

// MOTION/POUs/FBs/Basic/FB_MC2_AX5000
//------------------------------------------------------------------------------------------
//                                                                                        	
//***************************** Beckhoff TwinCAT Examples **********************************
//                                                                                        	
//************************************* WARNING ********************************************
// This program is only an example. If it is used as a control program in any real        	
// application, Beckhoff is not responsible for any malfunction, loss or damage           	
// which could arise by using this program!                                               	
//                                                                                        	
//*************************************  Program Info. *************************************
//                                                                                        	
// PLC program name:    	FB_MC2_AX5000 (FB)               	                           	
// Hardware platform:      	TwinCat PTP v3.1.4022				                          		                                  	
//                                                                                        	
// ======================================================================================== 
//         Version       Date                        Remarks                              	
// ======================================================================================== 
//         3.1           27 feb 2018                 First release of this example        	
// ======================================================================================== 
//                                                                                        	
//******************************* Aims OF this PLC PROGRAM *********************************
//                                                                                        	 
//                                                                                        	
//----------------------------------------------------------------------------------------- 
FUNCTION_BLOCK FB_MC2_AX5000 EXTENDS FB_MC2_Basic IMPLEMENTS I_MC2_AX5000
VAR
	FB_MC2_AX5000_M_nMC_Brake_bExecute: BOOL;
	FB_MC2_AX5000_M_nMC_Brake_eBrakeState: E_MC2_AX5000_Brake;
	FB_MC2_AX5000_M_nMC_Brake_iState: INT;
	FB_MC2_AX5000_M_nMC_Brake_nValue: UINT;
	FB_MC2_AX5000_M_nMC_Brake_fbExecute_R_TRIG: Tc2_Standard.R_TRIG;
	FB_MC2_AX5000_M_nMC_Brake_fbSoEWrite: TC2_MC2_DRIVE.FB_SoEWrite;

	FB_MC2_AX5000_M_nMC_ClrLagError_bExecute: BOOL;
	FB_MC2_AX5000_M_nMC_ClrLagError_iState: INT;
	FB_MC2_AX5000_M_nMC_ClrLagError_fbExecute_R_TRIG: Tc2_Standard.R_TRIG;
	FB_MC2_AX5000_M_nMC_ClrLagError_fbSoEWrite: TC2_MC2_DRIVE.FB_SoEWrite;
	FB_MC2_AX5000_M_nMC_ClrLagError_nData: UDINT;
	FB_MC2_AX5000_M_nMC_ClrLagError_bDone: BOOL;
	FB_MC2_AX5000_M_nMC_ClrLagError_nStatus: UDINT;

	FB_MC2_AX5000_M_nMC_DriveData_iState: INT;
	FB_MC2_AX5000_M_nMC_DriveData_fbSoEAX5000ReadActMainVoltage: FB_SoEAX5000ReadActMainVoltage;
	FB_MC2_AX5000_M_nMC_DriveData_fbSoEReadAmplifierTemperature: FB_SoEReadAmplifierTemperature;
	FB_MC2_AX5000_M_nMC_DriveData_fbSoEReadMotorTemperature: FB_SoEReadMotorTemperature;
	FB_MC2_AX5000_M_nMC_DriveData_fbSoERead: Tc2_MC2_Drive.FB_SoERead;
	FB_MC2_AX5000_M_nMC_DriveData_lrActualMainVoltage: LREAL;
	FB_MC2_AX5000_M_nMC_DriveData_lrAmplifierTemperature: LREAL;
	FB_MC2_AX5000_M_nMC_DriveData_lrMotorTemperature: LREAL;
	FB_MC2_AX5000_M_nMC_DriveData_nDiagnosticNumber: UDINT;

	FB_MC2_AX5000_M_nMC_MotorParam1_bExecute: BOOL;
	FB_MC2_AX5000_M_nMC_MotorParam1_bInverse: BOOL;
	FB_MC2_AX5000_M_nMC_MotorParam1_nMaxRpm: UINT;
	FB_MC2_AX5000_M_nMC_MotorParam1_lrDiameter: LREAL;
	FB_MC2_AX5000_M_nMC_MotorParam1_lrGearNumerator: LREAL;
	FB_MC2_AX5000_M_nMC_MotorParam1_lrGearDenominator: LREAL;
	FB_MC2_AX5000_M_nMC_MotorParam1_iState: INT;
	FB_MC2_AX5000_M_nMC_MotorParam1_fbExecute_R_TRIG: R_TRIG;
	FB_MC2_AX5000_M_nMC_MotorParam1_fbADSRDWRT: ADSRDWRT;
	FB_MC2_AX5000_M_nMC_MotorParam1_fbMC2_SetEncoderScalingFactor: MC_SetEncoderScalingFactor;
	FB_MC2_AX5000_M_nMC_MotorParam1_stMC2_Param: _ST_MC2_Param1;
	FB_MC2_AX5000_M_nMC_MotorParam1_arr_nADSReturn: ARRAY[1..6] OF UDINT;
	
	FB_MC2_AX5000_M_nMC_PID_PosCtrl_bExecute: BOOL;
	FB_MC2_AX5000_M_nMC_PID_PosCtrl_rKv: REAL; 
	FB_MC2_AX5000_M_nMC_PID_PosCtrl_iState: INT;
	FB_MC2_AX5000_M_nMC_PID_PosCtrl_iKv: INT;
	FB_MC2_AX5000_M_nMC_PID_PosCtrl_fbExecute_R_TRIG: R_TRIG;
	FB_MC2_AX5000_M_nMC_PID_PosCtrl_fbSoEWrite: TC2_MC2_DRIVE.FB_SoEWrite;

	FB_MC2_AX5000_M_nMC_Power_bEnable: BOOL;
	FB_MC2_AX5000_M_nMC_Power_bE_Stop: BOOL;
	FB_MC2_AX5000_M_nMC_Power_bE_StopDelay: BOOL;
	FB_MC2_AX5000_M_nMC_Power_bEnable_Positive: BOOL;
	FB_MC2_AX5000_M_nMC_Power_bEnable_Negative: BOOL;
	FB_MC2_AX5000_M_nMC_Power_fbStartDelay_TON: Tc2_Standard.TON;
	FB_MC2_AX5000_M_nMC_Power_arr_nRet: ARRAY[1..4] OF UDINT;
	
	FB_MC2_AX5000_M_nMC_Torque_bExecute: BOOL;
	FB_MC2_AX5000_M_nMC_Torque_lrTorque: LREAL; 		// Torque limit 0.0-100.0%	
	FB_MC2_AX5000_M_nMC_Torque_iState: INT;
	FB_MC2_AX5000_M_nMC_Torque_iTorque: INT;
	FB_MC2_AX5000_M_nMC_Torque_fbExecute_R_TRIG: R_TRIG;
	FB_MC2_AX5000_M_nMC_Torque_fbSoEWrite: TC2_MC2_DRIVE.FB_SoEWrite;
	
	FB_MC2_AX5000_M_nMC_TouchProbe1_bEnable: BOOL;
	FB_MC2_AX5000_M_nMC_TouchProbe1_lrPrellFilter_RisingEdge: LREAL;
	FB_MC2_AX5000_M_nMC_TouchProbe1_iState: INT;
	FB_MC2_AX5000_M_nMC_TouchProbe1_fbEnable_R_TRIG: R_TRIG;
	FB_MC2_AX5000_M_nMC_TouchProbe1_fbDisable_R_TRIG: R_TRIG;	
	FB_MC2_AX5000_M_nMC_TouchProbe1_fbTouchProbe: Tc2_MC2.MC_TouchProbe;
	FB_MC2_AX5000_M_nMC_TouchProbe1_fbAbortTrigger: Tc2_MC2.MC_AbortTrigger;
	FB_MC2_AX5000_M_nMC_TouchProbe1_stTriggerInput: Tc2_MC2.TRIGGER_REF;
	FB_MC2_AX5000_M_nMC_TouchProbe1_lrRecordedPosition1_RisingEdge: LREAL;
	FB_MC2_AX5000_M_nMC_TouchProbe1_lrLastLatchPosition: LREAL;

	FB_MC2_AX5000_M_nMC_TouchProbe2_bEnable: BOOL;
	FB_MC2_AX5000_M_nMC_TouchProbe2_bRisingEdgeDone: BOOL;
	FB_MC2_AX5000_M_nMC_TouchProbe2_iState: INT;
	FB_MC2_AX5000_M_nMC_TouchProbe2_lrPrellFilter_RisingEdge: LREAL;
	FB_MC2_AX5000_M_nMC_TouchProbe2_lrPrellFilter_FallingEdge: LREAL;
	FB_MC2_AX5000_M_nMC_TouchProbe2_fbEnable_R_TRIG: Tc2_Standard.R_TRIG;
	FB_MC2_AX5000_M_nMC_TouchProbe2_fbDisable_R_TRIG: Tc2_Standard.R_TRIG;	
	FB_MC2_AX5000_M_nMC_TouchProbe2_fbTouchProbe: Tc2_MC2.MC_TouchProbe;
	FB_MC2_AX5000_M_nMC_TouchProbe2_stTriggerInput: Tc2_MC2.TRIGGER_REF;
	FB_MC2_AX5000_M_nMC_TouchProbe2_fbAbortTrigger: Tc2_MC2.MC_AbortTrigger;
	FB_MC2_AX5000_M_nMC_TouchProbe2_lrRecordedPosition2_RisingEdge: LREAL;
	FB_MC2_AX5000_M_nMC_TouchProbe2_lrRecordedPosition2_FallingEdge: LREAL;
	FB_MC2_AX5000_M_nMC_TouchProbe2_lrLastLatchPosition: LREAL;
	
	FB_MC2_AX5000_M_nReset_iState: INT;
	FB_MC2_AX5000_M_nReset_fbExecute_R_TRIG: Tc2_Standard.R_TRIG;
	FB_MC2_AX5000_M_nReset_fbSoEReset: Tc2_MC2_Drive.FB_SoEReset;
	FB_MC2_AX5000_M_nReset_nStatus: UDINT;
END_VAR

//	The result of the method is an unsigned double integer
//	0 = idle 
//	1 = coupled
//	2 = starting
//	3 = running
//	4 = aborted
// 	5 = no hardware connected
// 	6 = Spare
//	7 = pointer or index error
//	8 = mapping error
//	9 = parameter error
//	10 = complete
//	Any other number = ErrorID
METHOD PUBLIC M_nMC_AcceptBlockedDriveSignal : UDINT
VAR_INPUT
	bExecute: BOOL;
END_VAR
// No hardware connected
IF NOT _bHardwareConnected THEN
	Tc2_MC2.MC_SetAcceptBlockedDriveSignal(Axis:= _stAXIS_REF, Enable:= FALSE);
	IF bExecute THEN
		M_nMC_AcceptBlockedDriveSignal:= Tc3_HBI_System.cNO_HARDWARE_CONNECTED;
	END_IF	
	RETURN;
END_IF

// Update function
IF _stAXIS_REF.NcToPlc.AxisID > 0 THEN
	IF _bHardwareConnected THEN
		IF Tc2_MC2.MC_SetAcceptBlockedDriveSignal(Axis:= _stAXIS_REF, Enable:= bExecute) THEN
			M_nMC_AcceptBlockedDriveSignal:= Tc3_HBI_System.cCOMPLETE;
		ELSE
			M_nMC_AcceptBlockedDriveSignal:= Tc3_HBI_System.cIDLE;
		END_IF	
	ELSE
		Tc2_MC2.MC_SetAcceptBlockedDriveSignal(Axis:= _stAXIS_REF, Enable:= FALSE);
		M_nMC_AcceptBlockedDriveSignal:= Tc3_HBI_System.cNO_HARDWARE_CONNECTED;
	END_IF
ELSE
	Tc2_MC2.MC_SetAcceptBlockedDriveSignal(Axis:= _stAXIS_REF, Enable:= FALSE); 
	IF bExecute THEN
		M_nMC_AcceptBlockedDriveSignal:= Tc3_HBI_System.cMAPPING_ERROR;		
	END_IF
	RETURN;
END_IF
END_METHOD

//	The result of the method is an unsigned double integer
//	0 = idle 
//	1 = coupled
//	2 = starting
//	3 = running
//	4 = aborted
// 	5 = no hardware connected
// 	6 = Spare
//	7 = pointer or index error
//	8 = mapping error
//	9 = parameter error
//	10 = complete
//	Any other number = ErrorID
METHOD PUBLIC M_nMC_Brake : UDINT
VAR_INPUT
	bExecute: BOOL;
	eBrakeState: E_MC2_AX5000_Brake;
END_VAR
// Local variable
FB_MC2_AX5000_M_nMC_Brake_bExecute:= bExecute;
FB_MC2_AX5000_M_nMC_Brake_eBrakeState:= eBrakeState;

//**********************************
// Reset 
//**********************************
IF _bReset THEN
	IF _bError THEN
		FB_MC2_AX5000_M_nMC_Brake_fbSoEWrite(Execute:= FALSE, Axis:= _stAXIS_REF); 
		FB_MC2_AX5000_M_nMC_Brake_iState:= 000;
	END_IF
END_IF

// No hardware connected
IF NOT _bHardwareConnected THEN
	FB_MC2_AX5000_M_nMC_Brake_fbSoEWrite(Execute:= FALSE, Axis:= _stAXIS_REF); 
	FB_MC2_AX5000_M_nMC_Brake_iState:= 000;
	IF FB_MC2_AX5000_M_nMC_Brake_bExecute THEN
		M_nMC_Brake:= Tc3_HBI_System.cNO_HARDWARE_CONNECTED;
	END_IF	
	RETURN;
END_IF

// Parameter check 
IF FB_MC2_AX5000_M_nMC_Brake_bExecute THEN
	IF FB_MC2_AX5000_M_nMC_Brake_eBrakeState = AX5000_Brake_Automatic OR FB_MC2_AX5000_M_nMC_Brake_eBrakeState = AX5000_Brake_Force_lock OR FB_MC2_AX5000_M_nMC_Brake_eBrakeState = AX5000_Brake_Force_unlock THEN
		;
	ELSE
		// Parameter error	
		M_nMC_Brake:= Tc3_HBI_System.cPARAMETER_ERROR;
		RETURN;
	END_IF
END_IF

//**********************************
// Wait for execute
//**********************************
IF _stAXIS_REF.NcToPlc.AxisID > 0 THEN
	FB_MC2_AX5000_M_nMC_Brake_fbExecute_R_TRIG(CLK:= FB_MC2_AX5000_M_nMC_Brake_bExecute);
	IF FB_MC2_AX5000_M_nMC_Brake_fbExecute_R_TRIG.Q THEN
		FB_MC2_AX5000_M_nMC_Brake_fbSoEWrite(Execute:= FALSE, Axis:= _stAXIS_REF); 
		FB_MC2_AX5000_M_nMC_Brake_iState:= 001;
	END_IF
ELSE
	FB_MC2_AX5000_M_nMC_Brake_fbSoEWrite(Execute:= FALSE, Axis:= _stAXIS_REF); 
	FB_MC2_AX5000_M_nMC_Brake_iState:= 000;
	IF FB_MC2_AX5000_M_nMC_Brake_bExecute THEN
		M_nMC_Brake:= Tc3_HBI_System.cMAPPING_ERROR;		
	END_IF
	RETURN;
END_IF


//**********************************
// Main sequence
//**********************************
CASE FB_MC2_AX5000_M_nMC_Brake_iState OF

	000: 	// Do nothing
	
	001:	// Set brake state
			M_nMC_Brake:= Tc3_HBI_System.cRUNNING;

			CASE FB_MC2_AX5000_M_nMC_Brake_eBrakeState OF
				
				AX5000_Brake_Automatic:
					FB_MC2_AX5000_M_nMC_Brake_nValue:= 0;

				AX5000_Brake_Force_lock:
					FB_MC2_AX5000_M_nMC_Brake_nValue:= 1;
			
				AX5000_Brake_Force_unlock:
					FB_MC2_AX5000_M_nMC_Brake_nValue:= 2;
				
			ELSE	
				FB_MC2_AX5000_M_nMC_Brake_nValue:= 0;
			END_CASE

			FB_MC2_AX5000_M_nMC_Brake_iState:= FB_MC2_AX5000_M_nMC_Brake_iState +1;

	002:	// Write brake state to AX5000
			M_nMC_Brake:= Tc3_HBI_System.cRUNNING;
			FB_MC2_AX5000_M_nMC_Brake_fbSoEWrite(Execute:= FALSE, Axis:= _stAXIS_REF); 
			FB_MC2_AX5000_M_nMC_Brake_fbSoEWrite(
				NetId:= '', 
				Idn:= P_0_IDN + 96, 
				Element:= 16#40, 
				pSrcBuf:= ADR(FB_MC2_AX5000_M_nMC_Brake_nValue), 
				BufLen:= SIZEOF(FB_MC2_AX5000_M_nMC_Brake_nValue), 
				Execute:= TRUE, 
				Timeout:= Tc2_System.DEFAULT_ADS_TIMEOUT, 
				Password:= , 
				Axis:= _stAXIS_REF, 
				Busy=> , 
				Error=> , 
				AdsErrId=> , 
				SercosErrId=> );
	
			FB_MC2_AX5000_M_nMC_Brake_iState:= FB_MC2_AX5000_M_nMC_Brake_iState +1;

	003:	// Write brake state
			M_nMC_Brake:= Tc3_HBI_System.cRUNNING;
			FB_MC2_AX5000_M_nMC_Brake_fbSoEWrite(Execute:= TRUE, Axis:= _stAXIS_REF); 
			
			// Error handling
			IF FB_MC2_AX5000_M_nMC_Brake_fbSoEWrite.Error THEN
				M_nError(FB_MC2_AX5000_M_nMC_Brake_fbSoEWrite.AdsErrId);
				M_nMC_Brake:= FB_MC2_AX5000_M_nMC_Brake_fbSoEWrite.AdsErrId;
			ELSE
				// Done
				IF NOT FB_MC2_AX5000_M_nMC_Brake_fbSoEWrite.Busy THEN
					FB_MC2_AX5000_M_nMC_Brake_fbSoEWrite(Execute:= FALSE, Axis:= _stAXIS_REF); 
					FB_MC2_AX5000_M_nMC_Brake_iState:= FB_MC2_AX5000_M_nMC_Brake_iState +1;
				END_IF	
			END_IF
		
	004:	// Done
			M_nMC_Brake:= Tc3_HBI_System.cCOMPLETE;
			IF NOT FB_MC2_AX5000_M_nMC_Brake_bExecute THEN
				FB_MC2_AX5000_M_nMC_Brake_iState:= 000;
			END_IF
			
ELSE
	FB_MC2_AX5000_M_nMC_Brake_iState:= 000;
END_CASE
END_METHOD

//	The result of the method is an unsigned double integer
//	0 = idle 
//	1 = coupled
//	2 = starting
//	3 = running
//	4 = aborted
// 	5 = no hardware connected
// 	6 = Spare
//	7 = pointer or index error
//	8 = mapping error
//	9 = parameter error
//	10 = complete
//	Any other number = ErrorID
METHOD PUBLIC M_nMC_ClrLagError : UDINT
VAR_INPUT
	bExecute: BOOL;
END_VAR
// Local varisble
FB_MC2_AX5000_M_nMC_ClrLagError_bExecute:= bExecute;

//**********************************
// Reset 
//**********************************
IF _bReset THEN
	IF _bError THEN
		FB_MC2_AX5000_M_nMC_ClrLagError_fbSoEWrite(Execute:= FALSE, Axis:= _stAXIS_REF); 
		SUPER^.M_nMC_ClrLagError(bExecute:= FALSE);
		FB_MC2_AX5000_M_nMC_ClrLagError_fbExecute_R_TRIG(CLK:= FALSE);
		FB_MC2_AX5000_M_nMC_ClrLagError_iState:= 000;
	END_IF
END_IF
// No hardware connected
IF NOT _bHardwareConnected THEN
	SUPER^.M_nMC_ClrLagError(bExecute:= FALSE);
	FB_MC2_AX5000_M_nMC_ClrLagError_fbExecute_R_TRIG(CLK:= FALSE);
	FB_MC2_AX5000_M_nMC_ClrLagError_iState:= 000;
	IF FB_MC2_AX5000_M_nMC_ClrLagError_bExecute THEN
		M_nMC_ClrLagError:= Tc3_HBI_System.cNO_HARDWARE_CONNECTED;
	END_IF	
	RETURN;
END_IF


//**********************************
// Wait for execute
//**********************************
IF _stAXIS_REF.NcToPlc.AxisID > 0 THEN
	FB_MC2_AX5000_M_nMC_ClrLagError_fbExecute_R_TRIG(CLK:= FB_MC2_AX5000_M_nMC_ClrLagError_bExecute);
	IF FB_MC2_AX5000_M_nMC_ClrLagError_fbExecute_R_TRIG.Q THEN
		FB_MC2_AX5000_M_nMC_ClrLagError_fbSoEWrite(Execute:= FALSE, Axis:= _stAXIS_REF); 
		SUPER^.M_nMC_ClrLagError(bExecute:= FALSE);
		IF FB_MC2_AX5000_M_nMC_ClrLagError_bDone THEN
			FB_MC2_AX5000_M_nMC_ClrLagError_iState:= 010;
		ELSE
			FB_MC2_AX5000_M_nMC_ClrLagError_iState:= 001;
		END_IF
	END_IF
ELSE
	FB_MC2_AX5000_M_nMC_ClrLagError_fbExecute_R_TRIG(CLK:= FALSE);
	FB_MC2_AX5000_M_nMC_ClrLagError_iState:= 000;
	IF FB_MC2_AX5000_M_nMC_ClrLagError_bExecute THEN
		M_nMC_ClrLagError:= Tc3_HBI_System.cMAPPING_ERROR;
	END_IF
	RETURN;
END_IF


//**********************************
// Main sequence
//**********************************
CASE FB_MC2_AX5000_M_nMC_ClrLagError_iState OF

	000: 	// Do nothing
	
	001:	// Reset lag error S_0_159 = 0	
			M_nMC_ClrLagError:= Tc3_HBI_System.cRUNNING;
			FB_MC2_AX5000_M_nMC_ClrLagError_nData:= 16#0000;
			FB_MC2_AX5000_M_nMC_ClrLagError_fbSoEWrite(Execute:= FALSE, Axis:= _stAXIS_REF); 
			FB_MC2_AX5000_M_nMC_ClrLagError_fbSoEWrite(
				NetId:= , 
				Idn:= S_0_IDN + 159, 
				Element:= 16#40, 
				pSrcBuf:= ADR(FB_MC2_AX5000_M_nMC_ClrLagError_nData), 
				BufLen:= SIZEOF(FB_MC2_AX5000_M_nMC_ClrLagError_nData), 
				Execute:= TRUE, 
				Timeout:= Tc2_System.DEFAULT_ADS_TIMEOUT, 
				Password:= , 
				Axis:= _stAXIS_REF, 
				Busy=> , 
				Error=> , 
				AdsErrId=> , 
				SercosErrId=> );
			
			FB_MC2_AX5000_M_nMC_ClrLagError_iState:= FB_MC2_AX5000_M_nMC_ClrLagError_iState +1;
	
	002:	// Reset Kv factor positions controller
			M_nMC_ClrLagError:= Tc3_HBI_System.cRUNNING;
			FB_MC2_AX5000_M_nMC_ClrLagError_fbSoEWrite(Execute:= TRUE, Axis:= _stAXIS_REF); 
	
			// Error handling
			IF FB_MC2_AX5000_M_nMC_ClrLagError_fbSoEWrite.Error THEN
				M_nError(FB_MC2_AX5000_M_nMC_ClrLagError_fbSoEWrite.AdsErrId);
				M_nMC_ClrLagError:= FB_MC2_AX5000_M_nMC_ClrLagError_fbSoEWrite.AdsErrId;
			ELSE
				// Done
				IF NOT FB_MC2_AX5000_M_nMC_ClrLagError_fbSoEWrite.Busy THEN
					FB_MC2_AX5000_M_nMC_ClrLagError_bDone:= TRUE;
					FB_MC2_AX5000_M_nMC_ClrLagError_fbSoEWrite(Execute:= FALSE, Axis:= _stAXIS_REF); 
					FB_MC2_AX5000_M_nMC_ClrLagError_iState:= 010;
				END_IF	
			END_IF

	010:	// Basic done
			M_nMC_ClrLagError:= SUPER^.M_nMC_ClrLagError(bExecute:= TRUE);			
			IF M_nMC_ClrLagError = Tc3_HBI_System.cCOMPLETE THEN
				SUPER^.M_nMC_ClrLagError(bExecute:= FALSE);
				FB_MC2_AX5000_M_nMC_ClrLagError_iState:= FB_MC2_AX5000_M_nMC_ClrLagError_iState +1;
			END_IF

	011:	// Done
			M_nMC_ClrLagError:= Tc3_HBI_System.cCOMPLETE;
			IF NOT FB_MC2_AX5000_M_nMC_ClrLagError_bExecute THEN
				FB_MC2_AX5000_M_nMC_ClrLagError_iState:= 000;
			END_IF
	
ELSE
	FB_MC2_AX5000_M_nMC_ClrLagError_iState:= 000;
END_CASE
END_METHOD

//	The result of the method is an unsigned double integer
//	0 = idle 
//	1 = coupled
//	2 = starting
//	3 = running
//	4 = aborted
// 	5 = no hardware connected
// 	6 = Spare
//	7 = pointer or index error
//	8 = mapping error
//	9 = parameter error
//	10 = complete
//	Any other number = ErrorID
METHOD PRIVATE M_nMC_DriveData : UDINT
//**********************************
// Reset 
//**********************************
IF _bReset THEN
	IF _bError THEN
		FB_MC2_AX5000_M_nMC_DriveData_fbSoEAX5000ReadActMainVoltage(Execute:= FALSE, Axis:= _stAXIS_REF);
		FB_MC2_AX5000_M_nMC_DriveData_fbSoEReadAmplifierTemperature(Execute:= FALSE, Axis:= _stAXIS_REF);
		FB_MC2_AX5000_M_nMC_DriveData_fbSoEReadMotorTemperature(Execute:= FALSE, Axis:= _stAXIS_REF); 
		FB_MC2_AX5000_M_nMC_DriveData_fbSoERead(Execute:= FALSE, Axis:= _stAXIS_REF); 
		FB_MC2_AX5000_M_nMC_DriveData_iState:= 000;
	END_IF
	RETURN;
END_IF

// No hardware connected
IF NOT _bHardwareConnected THEN
	FB_MC2_AX5000_M_nMC_DriveData_lrActualMainVoltage:= 0.0;		// Drive Main voltage
	FB_MC2_AX5000_M_nMC_DriveData_lrAmplifierTemperature:= 0.0;		// Drive temperatur
	FB_MC2_AX5000_M_nMC_DriveData_lrMotorTemperature:= 0.0;			// Motor temperatur
	FB_MC2_AX5000_M_nMC_DriveData_fbSoEAX5000ReadActMainVoltage(Execute:= FALSE, Axis:= _stAXIS_REF);
	FB_MC2_AX5000_M_nMC_DriveData_fbSoEReadAmplifierTemperature(Execute:= FALSE, Axis:= _stAXIS_REF);
	FB_MC2_AX5000_M_nMC_DriveData_fbSoEReadMotorTemperature(Execute:= FALSE, Axis:= _stAXIS_REF); 
	FB_MC2_AX5000_M_nMC_DriveData_iState:= 000;
	FB_MC2_AX5000_M_nMC_DriveData_fbSoERead(Execute:= FALSE, Axis:= _stAXIS_REF); 
	M_nMC_DriveData:= Tc3_HBI_System.cNO_HARDWARE_CONNECTED;
	RETURN;
END_IF

// Check for Axis
IF _stAXIS_REF.NcToPlc.AxisID = 0 THEN
	FB_MC2_AX5000_M_nMC_DriveData_fbSoEAX5000ReadActMainVoltage(Execute:= FALSE, Axis:= _stAXIS_REF);
	FB_MC2_AX5000_M_nMC_DriveData_fbSoEReadAmplifierTemperature(Execute:= FALSE, Axis:= _stAXIS_REF);
	FB_MC2_AX5000_M_nMC_DriveData_fbSoEReadMotorTemperature(Execute:= FALSE, Axis:= _stAXIS_REF); 
	FB_MC2_AX5000_M_nMC_DriveData_fbSoERead(Execute:= FALSE, Axis:= _stAXIS_REF); 
	FB_MC2_AX5000_M_nMC_DriveData_iState:= 000;
	RETURN;
END_IF

//**********************************
// Main sequence
//**********************************
CASE FB_MC2_AX5000_M_nMC_DriveData_iState OF

	000:	// Init
			M_nMC_DriveData:= Tc3_HBI_System.cSTARTING;
			FB_MC2_AX5000_M_nMC_DriveData_fbSoEAX5000ReadActMainVoltage(Execute:= FALSE, Axis:= _stAXIS_REF);
			FB_MC2_AX5000_M_nMC_DriveData_fbSoEReadAmplifierTemperature(Execute:= FALSE, Axis:= _stAXIS_REF);
			FB_MC2_AX5000_M_nMC_DriveData_fbSoEReadMotorTemperature(Execute:= FALSE, Axis:= _stAXIS_REF); 

			// Simulations axis 
			IF _stAXIS_REF.NcToPlc.AxisID > 0 THEN
				IF _stAXIS_REF.Status.OpMode.SimulationAxis THEN
					FB_MC2_AX5000_M_nMC_DriveData_lrActualMainVoltage:= 0.0;			// Drive Main voltage
					FB_MC2_AX5000_M_nMC_DriveData_lrAmplifierTemperature:= 0.0;		// Drive temperatur
					FB_MC2_AX5000_M_nMC_DriveData_lrMotorTemperature:= 0.0;			// Motor temperatur
					M_nMC_DriveData:= Tc3_HBI_System.cNO_HARDWARE_CONNECTED;
				ELSE
					// Axis connected to Hardware
					IF _bHardwareConnected THEN
						M_nMC_DriveData:= Tc3_HBI_System.cCOMPLETE;
						FB_MC2_AX5000_M_nMC_DriveData_iState:= FB_MC2_AX5000_M_nMC_DriveData_iState +1;
					ELSE
						FB_MC2_AX5000_M_nMC_DriveData_lrActualMainVoltage:= 0.0;		// Drive Main voltage
						FB_MC2_AX5000_M_nMC_DriveData_lrAmplifierTemperature:= 0.0;	// Drive temperatur
						FB_MC2_AX5000_M_nMC_DriveData_lrMotorTemperature:= 0.0;		// Motor temperatur
						M_nMC_DriveData:= Tc3_HBI_System.cNO_HARDWARE_CONNECTED;
					END_IF
				END_IF
			ELSE
				FB_MC2_AX5000_M_nMC_DriveData_lrActualMainVoltage:= 0.0;		// Drive Main voltage
				FB_MC2_AX5000_M_nMC_DriveData_lrAmplifierTemperature:= 0.0;	// Drive temperatur
				FB_MC2_AX5000_M_nMC_DriveData_lrMotorTemperature:= 0.0;		// Motor temperatur
				M_nMC_DriveData:= Tc3_HBI_System.cNO_HARDWARE_CONNECTED;
			END_IF
			
	001:	// Read actual main voltage
			M_nMC_DriveData:= Tc3_HBI_System.cCOMPLETE;
			FB_MC2_AX5000_M_nMC_DriveData_fbSoEAX5000ReadActMainVoltage(Execute:= TRUE, Axis:= _stAXIS_REF);
	
			// Error handling
			IF FB_MC2_AX5000_M_nMC_DriveData_fbSoEAX5000ReadActMainVoltage.Error THEN
				IF FB_MC2_AX5000_M_nMC_DriveData_fbSoEAX5000ReadActMainVoltage.AdsErrId <> 0 THEN
					M_nError(FB_MC2_AX5000_M_nMC_DriveData_fbSoEAX5000ReadActMainVoltage.AdsErrId);
					M_nMC_DriveData:= FB_MC2_AX5000_M_nMC_DriveData_fbSoEAX5000ReadActMainVoltage.AdsErrId;
				ELSE
					M_nError(FB_MC2_AX5000_M_nMC_DriveData_fbSoEAX5000ReadActMainVoltage.SercosErrId);
					M_nMC_DriveData:= FB_MC2_AX5000_M_nMC_DriveData_fbSoEAX5000ReadActMainVoltage.SercosErrId;
				END_IF
			ELSE
				// Done
				IF NOT FB_MC2_AX5000_M_nMC_DriveData_fbSoEAX5000ReadActMainVoltage.Busy THEN
					FB_MC2_AX5000_M_nMC_DriveData_fbSoEAX5000ReadActMainVoltage(Execute:= FALSE, Axis:= _stAXIS_REF);
					FB_MC2_AX5000_M_nMC_DriveData_lrActualMainVoltage:= FB_MC2_AX5000_M_nMC_DriveData_fbSoEAX5000ReadActMainVoltage.ActualMainVoltage;
					FB_MC2_AX5000_M_nMC_DriveData_iState:= FB_MC2_AX5000_M_nMC_DriveData_iState +1;
				END_IF	
			END_IF
	
	002:	// Read amplifier temperatur
			M_nMC_DriveData:= Tc3_HBI_System.cCOMPLETE;
			FB_MC2_AX5000_M_nMC_DriveData_fbSoEReadAmplifierTemperature(Execute:= TRUE, Axis:= _stAXIS_REF);
	
			// Error handling
			IF FB_MC2_AX5000_M_nMC_DriveData_fbSoEReadAmplifierTemperature.Error THEN
				IF FB_MC2_AX5000_M_nMC_DriveData_fbSoEReadAmplifierTemperature.AdsErrId <> 0 THEN
					M_nError(FB_MC2_AX5000_M_nMC_DriveData_fbSoEReadAmplifierTemperature.AdsErrId);
					M_nMC_DriveData:= FB_MC2_AX5000_M_nMC_DriveData_fbSoEReadAmplifierTemperature.AdsErrId;
				ELSE
					M_nError(FB_MC2_AX5000_M_nMC_DriveData_fbSoEReadAmplifierTemperature.SercosErrId);
					M_nMC_DriveData:= FB_MC2_AX5000_M_nMC_DriveData_fbSoEReadAmplifierTemperature.SercosErrId;
				END_IF
			ELSE
				// Done
				IF NOT FB_MC2_AX5000_M_nMC_DriveData_fbSoEReadAmplifierTemperature.Busy THEN
					FB_MC2_AX5000_M_nMC_DriveData_fbSoEReadAmplifierTemperature(Execute:= FALSE, Axis:= _stAXIS_REF);
					FB_MC2_AX5000_M_nMC_DriveData_lrAmplifierTemperature:= FB_MC2_AX5000_M_nMC_DriveData_fbSoEReadAmplifierTemperature.AmplifierTemperature;
					FB_MC2_AX5000_M_nMC_DriveData_iState:= FB_MC2_AX5000_M_nMC_DriveData_iState +1;
				END_IF	
			END_IF
	
	003:	// Read motor temperatur
			M_nMC_DriveData:= Tc3_HBI_System.cCOMPLETE;
			FB_MC2_AX5000_M_nMC_DriveData_fbSoEReadMotorTemperature(Execute:= TRUE, Axis:= _stAXIS_REF); 
			
			// Error handling
			IF FB_MC2_AX5000_M_nMC_DriveData_fbSoEReadMotorTemperature.Error THEN
				IF FB_MC2_AX5000_M_nMC_DriveData_fbSoEReadMotorTemperature.AdsErrId <> 0 THEN
					M_nError(FB_MC2_AX5000_M_nMC_DriveData_fbSoEReadMotorTemperature.AdsErrId);
					M_nMC_DriveData:= FB_MC2_AX5000_M_nMC_DriveData_fbSoEReadMotorTemperature.AdsErrId;
				ELSE
					M_nError(FB_MC2_AX5000_M_nMC_DriveData_fbSoEReadMotorTemperature.SercosErrId);
					M_nMC_DriveData:= FB_MC2_AX5000_M_nMC_DriveData_fbSoEReadMotorTemperature.SercosErrId;
				END_IF
			ELSE
				// Done
				IF NOT FB_MC2_AX5000_M_nMC_DriveData_fbSoEReadMotorTemperature.Busy THEN
					FB_MC2_AX5000_M_nMC_DriveData_fbSoEReadMotorTemperature(Execute:= FALSE, Axis:= _stAXIS_REF); 
					FB_MC2_AX5000_M_nMC_DriveData_lrMotorTemperature:= FB_MC2_AX5000_M_nMC_DriveData_fbSoEReadMotorTemperature.MotorTemperature;
					FB_MC2_AX5000_M_nMC_DriveData_iState:= FB_MC2_AX5000_M_nMC_DriveData_iState +1;
				END_IF	
			END_IF
	
	004:	// Read DiagnosticNumber
			M_nMC_DriveData:= Tc3_HBI_System.cCOMPLETE;
			FB_MC2_AX5000_M_nMC_DriveData_fbSoERead(
				NetId:= '', 
				Idn:= S_0_IDN + 390, 
				Element:= 16#40, 
				pDstBuf:= ADR(FB_MC2_AX5000_M_nMC_DriveData_nDiagnosticNumber), 
				BufLen:= SIZEOF(FB_MC2_AX5000_M_nMC_DriveData_nDiagnosticNumber), 
				Execute:= TRUE, 
				Timeout:= Tc2_System.DEFAULT_ADS_TIMEOUT, 
				Axis:= _stAXIS_REF, 
				Busy=> , 
				Error=> , 
				AdsErrId=> , 
				SercosErrId=> , 
				Attribute=> );
			
			// Error handling
			IF FB_MC2_AX5000_M_nMC_DriveData_fbSoERead.Error THEN
				IF FB_MC2_AX5000_M_nMC_DriveData_fbSoERead.AdsErrId <> 0 THEN
					M_nError(FB_MC2_AX5000_M_nMC_DriveData_fbSoERead.AdsErrId);
					M_nMC_DriveData:= FB_MC2_AX5000_M_nMC_DriveData_fbSoERead.AdsErrId;
				ELSE
					M_nError(FB_MC2_AX5000_M_nMC_DriveData_fbSoERead.SercosErrId);
					M_nMC_DriveData:= FB_MC2_AX5000_M_nMC_DriveData_fbSoERead.SercosErrId;
				END_IF
			ELSE
				// Done
				IF NOT FB_MC2_AX5000_M_nMC_DriveData_fbSoERead.Busy THEN
					FB_MC2_AX5000_M_nMC_DriveData_fbSoERead(Execute:= FALSE, Axis:= _stAXIS_REF); 
					FB_MC2_AX5000_M_nMC_DriveData_iState:= FB_MC2_AX5000_M_nMC_DriveData_iState +1;
				END_IF	
			END_IF

	005:	// Done
			M_nMC_DriveData:= Tc3_HBI_System.cCOMPLETE;
			FB_MC2_AX5000_M_nMC_DriveData_iState:= 000;
	
ELSE
	FB_MC2_AX5000_M_nMC_DriveData_iState:= 000;
END_CASE
END_METHOD

//	The result of the method is an unsigned double integer
//	0 = idle 
//	1 = coupled
//	2 = starting
//	3 = running
//	4 = aborted
// 	5 = no hardware connected
// 	6 = Spare
//	7 = pointer or index error
//	8 = mapping error
//	9 = parameter error
//	10 = complete
//	Any other number = ErrorID
METHOD PUBLIC M_nMC_MotorParam1 : UDINT
VAR_INPUT
	bExecute: BOOL;
	bInverse: BOOL;
	nMaxRpm: UINT;
	lrDiameter: LREAL;
	lrGearNumerator: LREAL;
	lrGearDenominator: LREAL;
END_VAR
// Local variable
FB_MC2_AX5000_M_nMC_MotorParam1_bExecute:= bExecute;
FB_MC2_AX5000_M_nMC_MotorParam1_bInverse:= bInverse;
FB_MC2_AX5000_M_nMC_MotorParam1_nMaxRpm:= nMaxRpm;
FB_MC2_AX5000_M_nMC_MotorParam1_lrDiameter:= lrDiameter;
FB_MC2_AX5000_M_nMC_MotorParam1_lrGearNumerator:= lrGearNumerator;
FB_MC2_AX5000_M_nMC_MotorParam1_lrGearDenominator:= lrGearDenominator;

//**********************************
// Reset 
//**********************************
IF _bReset THEN
	IF _bError THEN
		FB_MC2_AX5000_M_nMC_MotorParam1_fbADSRDWRT(WRTRD:= FALSE); 
		FB_MC2_AX5000_M_nMC_MotorParam1_fbMC2_SetEncoderScalingFactor(Axis:= _stAXIS_REF, Execute:= FALSE);
		FB_MC2_AX5000_M_nMC_MotorParam1_fbExecute_R_TRIG(CLK:= FALSE);
		FB_MC2_AX5000_M_nMC_MotorParam1_iState:= 000;
	END_IF
END_IF
// No hardware connected
IF NOT _bHardwareConnected THEN
	FB_MC2_AX5000_M_nMC_MotorParam1_fbADSRDWRT(WRTRD:= FALSE); 
	FB_MC2_AX5000_M_nMC_MotorParam1_fbMC2_SetEncoderScalingFactor(Axis:= _stAXIS_REF, Execute:= FALSE);
	FB_MC2_AX5000_M_nMC_MotorParam1_fbExecute_R_TRIG(CLK:= FALSE);
	FB_MC2_AX5000_M_nMC_MotorParam1_iState:= 000;
	IF FB_MC2_AX5000_M_nMC_MotorParam1_bExecute THEN
		M_nMC_MotorParam1:= Tc3_HBI_System.cNO_HARDWARE_CONNECTED;
	END_IF
	RETURN;
END_IF

//**********************************
// Parameter check 
//**********************************
IF FB_MC2_AX5000_M_nMC_MotorParam1_bExecute THEN
	IF FB_MC2_AX5000_M_nMC_MotorParam1_nMaxRpm <= 0.0 OR FB_MC2_AX5000_M_nMC_MotorParam1_lrDiameter <= 0.0 OR FB_MC2_AX5000_M_nMC_MotorParam1_lrGearNumerator <= 0.0 OR FB_MC2_AX5000_M_nMC_MotorParam1_lrGearDenominator <= 0.0 THEN
		M_nMC_MotorParam1:= Tc3_HBI_System.cPARAMETER_ERROR;

		FB_MC2_AX5000_M_nMC_MotorParam1_fbADSRDWRT(WRTRD:= FALSE); 
		FB_MC2_AX5000_M_nMC_MotorParam1_fbMC2_SetEncoderScalingFactor(Axis:= _stAXIS_REF, Execute:= FALSE);
		FB_MC2_AX5000_M_nMC_MotorParam1_fbExecute_R_TRIG(CLK:= FALSE);
		FB_MC2_AX5000_M_nMC_MotorParam1_iState:= 000;
		RETURN;
	END_IF
END_IF

	
//**********************************
// Wait for execute
//**********************************
IF _stAXIS_REF.NcToPlc.AxisID > 0 THEN
	FB_MC2_AX5000_M_nMC_MotorParam1_fbExecute_R_TRIG(CLK:= FB_MC2_AX5000_M_nMC_MotorParam1_bExecute);
	IF FB_MC2_AX5000_M_nMC_MotorParam1_fbExecute_R_TRIG.Q THEN
		FB_MC2_AX5000_M_nMC_MotorParam1_fbADSRDWRT(WRTRD:= FALSE); 
		FB_MC2_AX5000_M_nMC_MotorParam1_fbMC2_SetEncoderScalingFactor(Axis:= _stAXIS_REF, Execute:= FALSE);
		
		// Axis not coupled	
		IF NOT _stAXIS_REF.Status.Coupled THEN
			FB_MC2_AX5000_M_nMC_MotorParam1_iState:= 001;
		ELSE
			FB_MC2_AX5000_M_nMC_MotorParam1_iState:= 010;
		END_IF
	
	END_IF
ELSE
	FB_MC2_AX5000_M_nMC_MotorParam1_fbExecute_R_TRIG(CLK:= FALSE);
	FB_MC2_AX5000_M_nMC_MotorParam1_iState:= 000;
	IF FB_MC2_AX5000_M_nMC_MotorParam1_bExecute THEN
		M_nMC_MotorParam1:= Tc3_HBI_System.cMAPPING_ERROR;
	END_IF
	RETURN;
END_IF


//**********************************
// Main sequence
//**********************************
CASE FB_MC2_AX5000_M_nMC_MotorParam1_iState OF

	000: 	// Do nothing
	
	001:	// Check parameter input
			M_nMC_MotorParam1:= Tc3_HBI_System.cRUNNING;
			IF FB_MC2_AX5000_M_nMC_MotorParam1_nMaxRpm > 0.0 AND FB_MC2_AX5000_M_nMC_MotorParam1_lrDiameter > 0.0 AND FB_MC2_AX5000_M_nMC_MotorParam1_lrGearDenominator > 0.0 AND FB_MC2_AX5000_M_nMC_MotorParam1_lrGearNumerator > 0.0 THEN 
				FB_MC2_AX5000_M_nMC_MotorParam1_iState:= 2;
			ELSE
				M_nMC_MotorParam1:= Tc3_HBI_System.cPARAMETER_ERROR;
				IF NOT FB_MC2_AX5000_M_nMC_MotorParam1_bExecute THEN
					FB_MC2_AX5000_M_nMC_MotorParam1_iState:= 000;
				END_IF
			END_IF

	002:	// Parameter setup
			M_nMC_MotorParam1:= Tc3_HBI_System.cRUNNING;
		
			(* Copy values to transfer *)
			FB_MC2_AX5000_M_nMC_MotorParam1_stMC2_Param.nEncoderDir:= BOOL_TO_WORD(FB_MC2_AX5000_M_nMC_MotorParam1_bInverse);
			FB_MC2_AX5000_M_nMC_MotorParam1_stMC2_Param.nMotorDir:= BOOL_TO_WORD(FB_MC2_AX5000_M_nMC_MotorParam1_bInverse);
			FB_MC2_AX5000_M_nMC_MotorParam1_stMC2_Param.nHomeCamDir:= BOOL_TO_WORD( FB_MC2_AX5000_M_nMC_MotorParam1_bInverse);
			FB_MC2_AX5000_M_nMC_MotorParam1_stMC2_Param.nHomeSyncDir:= BOOL_TO_WORD(NOT FB_MC2_AX5000_M_nMC_MotorParam1_bInverse);
			FB_MC2_AX5000_M_nMC_MotorParam1_stMC2_Param.lrMaxVelocity:= (FB_MC2_AX5000_M_nMC_MotorParam1_nMaxRpm / 60.0) * (((FB_MC2_AX5000_M_nMC_MotorParam1_lrDiameter * PI) * FB_MC2_AX5000_M_nMC_MotorParam1_lrGearNumerator) / FB_MC2_AX5000_M_nMC_MotorParam1_lrGearDenominator);
			FB_MC2_AX5000_M_nMC_MotorParam1_stMC2_Param.lrRefVelocity:= FB_MC2_AX5000_M_nMC_MotorParam1_stMC2_Param.lrMaxVelocity * 1.1;
		
			// Setup adresses for transfer - The lines must be in the same order as the struct
			_iIdx:= 1;
			FB_MC2_AX5000_M_nMC_MotorParam1_stMC2_Param.aParm[_iIdx].nIndexGroup:= 16#00005000 + _stAXIS_REF.NcToPlc.AxisId; 	FB_MC2_AX5000_M_nMC_MotorParam1_stMC2_Param.aParm[_iIdx].nIndexOffset:= 16#00000008;	FB_MC2_AX5000_M_nMC_MotorParam1_stMC2_Param.aParm[_iIdx].nDataSize:= SIZEOF(FB_MC2_AX5000_M_nMC_MotorParam1_stMC2_Param.nEncoderDir);		_iIdx := _iIdx+1;
			FB_MC2_AX5000_M_nMC_MotorParam1_stMC2_Param.aParm[_iIdx].nIndexGroup:= 16#00007000 + _stAXIS_REF.NcToPlc.AxisId; 	FB_MC2_AX5000_M_nMC_MotorParam1_stMC2_Param.aParm[_iIdx].nIndexOffset:= 16#00000006;	FB_MC2_AX5000_M_nMC_MotorParam1_stMC2_Param.aParm[_iIdx].nDataSize:= SIZEOF(FB_MC2_AX5000_M_nMC_MotorParam1_stMC2_Param.nMotorDir);			_iIdx := _iIdx+1;
			FB_MC2_AX5000_M_nMC_MotorParam1_stMC2_Param.aParm[_iIdx].nIndexGroup:= 16#00005000 + _stAXIS_REF.NcToPlc.AxisId; 	FB_MC2_AX5000_M_nMC_MotorParam1_stMC2_Param.aParm[_iIdx].nIndexOffset:= 16#00000101;	FB_MC2_AX5000_M_nMC_MotorParam1_stMC2_Param.aParm[_iIdx].nDataSize:= SIZEOF(FB_MC2_AX5000_M_nMC_MotorParam1_stMC2_Param.nHomeCamDir);		_iIdx := _iIdx+1;
			FB_MC2_AX5000_M_nMC_MotorParam1_stMC2_Param.aParm[_iIdx].nIndexGroup:= 16#00005000 + _stAXIS_REF.NcToPlc.AxisId; 	FB_MC2_AX5000_M_nMC_MotorParam1_stMC2_Param.aParm[_iIdx].nIndexOffset:= 16#00000102;	FB_MC2_AX5000_M_nMC_MotorParam1_stMC2_Param.aParm[_iIdx].nDataSize:= SIZEOF(FB_MC2_AX5000_M_nMC_MotorParam1_stMC2_Param.nHomeSyncDir);		_iIdx := _iIdx+1;
			FB_MC2_AX5000_M_nMC_MotorParam1_stMC2_Param.aParm[_iIdx].nIndexGroup:= 16#00007000 + _stAXIS_REF.NcToPlc.AxisId; 	FB_MC2_AX5000_M_nMC_MotorParam1_stMC2_Param.aParm[_iIdx].nIndexOffset:= 16#00000101;	FB_MC2_AX5000_M_nMC_MotorParam1_stMC2_Param.aParm[_iIdx].nDataSize:= SIZEOF(FB_MC2_AX5000_M_nMC_MotorParam1_stMC2_Param.lrRefVelocity);		_iIdx := _iIdx+1;
			FB_MC2_AX5000_M_nMC_MotorParam1_stMC2_Param.aParm[_iIdx].nIndexGroup:= 16#00004000 + _stAXIS_REF.NcToPlc.AxisId; 	FB_MC2_AX5000_M_nMC_MotorParam1_stMC2_Param.aParm[_iIdx].nIndexOffset:= 16#00000027;	FB_MC2_AX5000_M_nMC_MotorParam1_stMC2_Param.aParm[_iIdx].nDataSize:= SIZEOF(FB_MC2_AX5000_M_nMC_MotorParam1_stMC2_Param.lrMaxVelocity);		_iIdx := _iIdx+1;
			
			FB_MC2_AX5000_M_nMC_MotorParam1_iState:= 003;
		
	003:	// Write ADS list 
			M_nMC_MotorParam1:= Tc3_HBI_System.cRUNNING;
			FB_MC2_AX5000_M_nMC_MotorParam1_fbADSRDWRT(WRTRD:= FALSE); 
			FB_MC2_AX5000_M_nMC_MotorParam1_fbADSRDWRT(
				NETID:= '', 
				PORT:= 501,
				IDXGRP:= 16#F081, 	// Write list 
				IDXOFFS:= SIZEOF(FB_MC2_AX5000_M_nMC_MotorParam1_arr_nADSReturn) / SIZEOF(FB_MC2_AX5000_M_nMC_MotorParam1_arr_nADSReturn[1]),
				WRITELEN:= SIZEOF(FB_MC2_AX5000_M_nMC_MotorParam1_stMC2_Param),
				READLEN:= SIZEOF(FB_MC2_AX5000_M_nMC_MotorParam1_arr_nADSReturn),
				SRCADDR:= ADR(FB_MC2_AX5000_M_nMC_MotorParam1_stMC2_Param),
				DESTADDR:= ADR(FB_MC2_AX5000_M_nMC_MotorParam1_arr_nADSReturn),
				WRTRD:= TRUE, 
				TMOUT:= T#2S); 
	
			FB_MC2_AX5000_M_nMC_MotorParam1_iState:= 004;
	
	004:	// Done		
			M_nMC_MotorParam1:= Tc3_HBI_System.cRUNNING;
			FB_MC2_AX5000_M_nMC_MotorParam1_fbADSRDWRT(WRTRD:= TRUE); 
				
			// Error handling
			IF FB_MC2_AX5000_M_nMC_MotorParam1_fbADSRDWRT.ERR THEN
				M_nError(FB_MC2_AX5000_M_nMC_MotorParam1_fbADSRDWRT.ERRID);
				M_nMC_MotorParam1:= FB_MC2_AX5000_M_nMC_MotorParam1_fbADSRDWRT.ERRID;
			ELSE
				// Done
				IF NOT FB_MC2_AX5000_M_nMC_MotorParam1_fbADSRDWRT.BUSY THEN
					FB_MC2_AX5000_M_nMC_MotorParam1_fbADSRDWRT(WRTRD:= FALSE); 
					FB_MC2_AX5000_M_nMC_MotorParam1_iState:= 005;
				END_IF
			END_IF

	005:	// Write list error handling
			M_nMC_MotorParam1:= Tc3_HBI_System.cRUNNING;
			FOR _iIdx := 1 TO UDINT_TO_INT(FB_MC2_AX5000_M_nMC_MotorParam1_fbADSRDWRT.IDXOFFS) DO
				IF _bError = FALSE THEN
					IF (FB_MC2_AX5000_M_nMC_MotorParam1_arr_nADSReturn[_iIdx] <> 0) THEN
						M_nError(nErrorID:= FB_MC2_AX5000_M_nMC_MotorParam1_arr_nADSReturn[_iIdx]);
						M_nMC_MotorParam1:= FB_MC2_AX5000_M_nMC_MotorParam1_arr_nADSReturn[_iIdx];
					END_IF
				END_IF
			END_FOR
			FB_MC2_AX5000_M_nMC_MotorParam1_iState:= 006;
		
	006:	// Write list error handling	
			M_nMC_MotorParam1:= Tc3_HBI_System.cRUNNING;
			IF NOT _bError THEN
				FB_MC2_AX5000_M_nMC_MotorParam1_iState:= 007;
			ELSE
				M_nMC_MotorParam1:= _nErrorID;
				IF NOT FB_MC2_AX5000_M_nMC_MotorParam1_bExecute THEN
					FB_MC2_AX5000_M_nMC_MotorParam1_iState:= 000;
				END_IF
			END_IF
	
	007:	// Write scale factor
			M_nMC_MotorParam1:= Tc3_HBI_System.cRUNNING;
			FB_MC2_AX5000_M_nMC_MotorParam1_fbMC2_SetEncoderScalingFactor(Axis:= _stAXIS_REF, Execute:= FALSE);
			FB_MC2_AX5000_M_nMC_MotorParam1_fbMC2_SetEncoderScalingFactor(
				Axis:= _stAXIS_REF, 
				Execute:= TRUE, 
				ScalingFactor:= (((FB_MC2_AX5000_M_nMC_MotorParam1_lrDiameter * PI) * FB_MC2_AX5000_M_nMC_MotorParam1_lrGearNumerator) / FB_MC2_AX5000_M_nMC_MotorParam1_lrGearDenominator) / (16#000FFFFF +1)); 
	
			FB_MC2_AX5000_M_nMC_MotorParam1_iState:= 008;
			
	008:	// Done
			M_nMC_MotorParam1:= Tc3_HBI_System.cRUNNING;
			FB_MC2_AX5000_M_nMC_MotorParam1_fbMC2_SetEncoderScalingFactor(Axis:= _stAXIS_REF, Execute:= TRUE);
		
			// Error handling
			IF FB_MC2_AX5000_M_nMC_MotorParam1_fbMC2_SetEncoderScalingFactor.Error THEN
				M_nError(nErrorID:= FB_MC2_AX5000_M_nMC_MotorParam1_fbMC2_SetEncoderScalingFactor.ErrorID);
				M_nMC_MotorParam1:= FB_MC2_AX5000_M_nMC_MotorParam1_fbMC2_SetEncoderScalingFactor.ErrorID;
			ELSE
				// Done
				IF FB_MC2_AX5000_M_nMC_MotorParam1_fbMC2_SetEncoderScalingFactor.Done THEN
					FB_MC2_AX5000_M_nMC_MotorParam1_fbMC2_SetEncoderScalingFactor(Axis:= _stAXIS_REF, Execute:= FALSE);
					FB_MC2_AX5000_M_nMC_MotorParam1_iState:= 020;
				END_IF
			END_IF
		
	010:	// Coupled
			M_nMC_MotorParam1:= Tc3_HBI_System.cCOUPLED;
			IF NOT FB_MC2_AX5000_M_nMC_MotorParam1_bExecute THEN
				FB_MC2_AX5000_M_nMC_MotorParam1_fbADSRDWRT(WRTRD:= FALSE); 
				FB_MC2_AX5000_M_nMC_MotorParam1_fbMC2_SetEncoderScalingFactor(Axis:= _stAXIS_REF, Execute:= FALSE);
				FB_MC2_AX5000_M_nMC_MotorParam1_iState:= 000;
			END_IF	

	020:	// Done
			M_nMC_MotorParam1:= Tc3_HBI_System.cCOMPLETE;
			IF NOT FB_MC2_AX5000_M_nMC_MotorParam1_bExecute THEN
				FB_MC2_AX5000_M_nMC_MotorParam1_fbADSRDWRT(WRTRD:= FALSE); 
				FB_MC2_AX5000_M_nMC_MotorParam1_fbMC2_SetEncoderScalingFactor(Axis:= _stAXIS_REF, Execute:= FALSE);
				FB_MC2_AX5000_M_nMC_MotorParam1_iState:= 000;
			END_IF	
		
ELSE
	FB_MC2_AX5000_M_nMC_MotorParam1_iState:= 000;
END_CASE
END_METHOD

//	The result of the method is an unsigned double integer
//	0 = idle 
//	1 = coupled
//	2 = starting
//	3 = running
//	4 = aborted
// 	5 = no hardware connected
// 	6 = Spare
//	7 = pointer or index error
//	8 = mapping error
//	9 = parameter error
//	10 = complete
//	Any other number = ErrorID
METHOD PUBLIC M_nMC_PID_PosCtrl : UDINT
VAR_INPUT
	bExecute: BOOL;
	rKv: REAL; 
END_VAR
// Local variable
FB_MC2_AX5000_M_nMC_PID_PosCtrl_bExecute:= bExecute;
FB_MC2_AX5000_M_nMC_PID_PosCtrl_rKv:= rKv;

//**********************************
// Reset 
//**********************************
IF _bReset THEN
	IF _bError THEN
		FB_MC2_AX5000_M_nMC_PID_PosCtrl_fbSoEWrite(Execute:= FALSE, Axis:= _stAXIS_REF);
		FB_MC2_AX5000_M_nMC_PID_PosCtrl_fbExecute_R_TRIG(CLK:= FALSE);
		FB_MC2_AX5000_M_nMC_PID_PosCtrl_iState:= 000;
	END_IF
END_IF
// No hardware connected
IF NOT _bHardwareConnected THEN
	FB_MC2_AX5000_M_nMC_PID_PosCtrl_fbSoEWrite(Execute:= FALSE, Axis:= _stAXIS_REF);
	FB_MC2_AX5000_M_nMC_PID_PosCtrl_fbExecute_R_TRIG(CLK:= FALSE);
	FB_MC2_AX5000_M_nMC_PID_PosCtrl_iState:= 000;
	IF FB_MC2_AX5000_M_nMC_PID_PosCtrl_bExecute THEN
		M_nMC_PID_PosCtrl:= Tc3_HBI_System.cNO_HARDWARE_CONNECTED;
	END_IF	
	RETURN;
END_IF

//**********************************
// Parameter check 
//**********************************
IF FB_MC2_AX5000_M_nMC_PID_PosCtrl_bExecute THEN
	IF FB_MC2_AX5000_M_nMC_PID_PosCtrl_rKv < 0.0 OR FB_MC2_AX5000_M_nMC_PID_PosCtrl_rKv > 100.0 THEN
		M_nMC_PID_PosCtrl:= Tc3_HBI_System.cPARAMETER_ERROR;

		FB_MC2_AX5000_M_nMC_PID_PosCtrl_fbSoEWrite(Execute:= FALSE, Axis:= _stAXIS_REF);
		FB_MC2_AX5000_M_nMC_PID_PosCtrl_fbExecute_R_TRIG(CLK:= FALSE);
		FB_MC2_AX5000_M_nMC_PID_PosCtrl_iState:= 000;
		RETURN;
	END_IF
END_IF


//**********************************
// Wait for execute
//**********************************
IF _stAXIS_REF.NcToPlc.AxisID > 0 THEN
	FB_MC2_AX5000_M_nMC_PID_PosCtrl_fbExecute_R_TRIG(CLK:= FB_MC2_AX5000_M_nMC_PID_PosCtrl_bExecute);
	IF FB_MC2_AX5000_M_nMC_PID_PosCtrl_fbExecute_R_TRIG.Q THEN
		FB_MC2_AX5000_M_nMC_PID_PosCtrl_fbSoEWrite(Execute:= FALSE, Axis:= _stAXIS_REF); 
		FB_MC2_AX5000_M_nMC_PID_PosCtrl_iState:= 001;
	END_IF
ELSE
	FB_MC2_AX5000_M_nMC_PID_PosCtrl_fbExecute_R_TRIG(CLK:= FALSE);
	FB_MC2_AX5000_M_nMC_PID_PosCtrl_iState:= 000;
	IF bExecute THEN
		M_nMC_PID_PosCtrl:= Tc3_HBI_System.cMAPPING_ERROR;
	END_IF
	RETURN;
END_IF


//**********************************
// Main sequence
//**********************************
CASE FB_MC2_AX5000_M_nMC_PID_PosCtrl_iState OF

	000: 	// Do nothing
	
	001:	// Reset Kv factor positions controller	
			M_nMC_PID_PosCtrl:= Tc3_HBI_System.cRUNNING;
			FB_MC2_AX5000_M_nMC_PID_PosCtrl_iKv:= REAL_TO_INT(FB_MC2_AX5000_M_nMC_PID_PosCtrl_rKv * 100.0);
			FB_MC2_AX5000_M_nMC_PID_PosCtrl_fbSoEWrite(Execute:= FALSE, Axis:= _stAXIS_REF); 
			FB_MC2_AX5000_M_nMC_PID_PosCtrl_fbSoEWrite(
				NetId:= , 
				Idn:= S_0_IDN + 104, 
				Element:= 16#40, 
				pSrcBuf:= ADR(FB_MC2_AX5000_M_nMC_PID_PosCtrl_iKv), 
				BufLen:= SIZEOF(FB_MC2_AX5000_M_nMC_PID_PosCtrl_iKv), 
				Execute:= TRUE, 
				Timeout:= Tc2_System.DEFAULT_ADS_TIMEOUT, 
				Password:= , 
				Axis:= _stAXIS_REF, 
				Busy=> , 
				Error=> , 
				AdsErrId=> , 
				SercosErrId=> );
			
			FB_MC2_AX5000_M_nMC_PID_PosCtrl_iState:= FB_MC2_AX5000_M_nMC_PID_PosCtrl_iState +1;
	
	002:	// Reset Kv factor positions controller
			M_nMC_PID_PosCtrl:= Tc3_HBI_System.cRUNNING;
			FB_MC2_AX5000_M_nMC_PID_PosCtrl_fbSoEWrite(Execute:= TRUE, Axis:= _stAXIS_REF); 
	
			// Error handling
			IF FB_MC2_AX5000_M_nMC_PID_PosCtrl_fbSoEWrite.Error THEN
				M_nError(FB_MC2_AX5000_M_nMC_PID_PosCtrl_fbSoEWrite.AdsErrId);
				M_nMC_PID_PosCtrl:= FB_MC2_AX5000_M_nMC_PID_PosCtrl_fbSoEWrite.AdsErrId;
			ELSE
				// Done
				IF NOT FB_MC2_AX5000_M_nMC_PID_PosCtrl_fbSoEWrite.Busy THEN
					FB_MC2_AX5000_M_nMC_PID_PosCtrl_fbSoEWrite(Execute:= FALSE, Axis:= _stAXIS_REF); 
					FB_MC2_AX5000_M_nMC_PID_PosCtrl_iState:= FB_MC2_AX5000_M_nMC_PID_PosCtrl_iState +1;
				END_IF	
			END_IF

	003:	// Done
			M_nMC_PID_PosCtrl:= Tc3_HBI_System.cCOMPLETE;
			IF NOT FB_MC2_AX5000_M_nMC_PID_PosCtrl_bExecute THEN
				FB_MC2_AX5000_M_nMC_PID_PosCtrl_iState:= 000;
			END_IF
	
ELSE
	FB_MC2_AX5000_M_nMC_PID_PosCtrl_iState:= 000;
END_CASE
END_METHOD

//	The result of the method is an unsigned double integer
//	0 = idle 
//	1 = coupled
//	2 = starting
//	3 = running
//	4 = aborted
// 	5 = no hardware connected
// 	6 = Spare
//	7 = pointer or index error
//	8 = mapping error
//	9 = parameter error
//	10 = complete
//	Any other number = ErrorID
METHOD PUBLIC M_nMC_Power : UDINT
VAR_INPUT
	bEnable: BOOL;
	bE_Stop: BOOL;
	bE_StopDelay: BOOL;
	bEnable_Positive: BOOL;
	bEnable_Negative: BOOL;
END_VAR
// Local variable
FB_MC2_AX5000_M_nMC_Power_bEnable:= bEnable;
FB_MC2_AX5000_M_nMC_Power_bE_Stop:= bE_Stop;
FB_MC2_AX5000_M_nMC_Power_bE_StopDelay:= bE_StopDelay; 
FB_MC2_AX5000_M_nMC_Power_bEnable_Positive:= bEnable_Positive;
FB_MC2_AX5000_M_nMC_Power_bEnable_Negative:= bEnable_Negative;

//**********************************
// Reset 
//**********************************
IF _bReset THEN
	MEMSET(destAddr:= ADR(FB_MC2_AX5000_M_nMC_Power_arr_nRet), fillByte:= 16#00, n:= SIZEOF(FB_MC2_AX5000_M_nMC_Power_arr_nRet));

	M_nMC_Brake(bExecute:= FB_MC2_AX5000_M_nMC_Brake_bExecute, eBrakeState:= FB_MC2_AX5000_M_nMC_Brake_eBrakeState);	
	M_nMC_ClrLagError(bExecute:= FB_MC2_AX5000_M_nMC_ClrLagError_bExecute);
	M_nMC_DriveData();
	M_nMC_MotorParam1(bExecute:= FB_MC2_AX5000_M_nMC_MotorParam1_bExecute, bInverse:= FB_MC2_AX5000_M_nMC_MotorParam1_bInverse,nMaxRpm:= FB_MC2_AX5000_M_nMC_MotorParam1_nMaxRpm,lrDiameter:= FB_MC2_AX5000_M_nMC_MotorParam1_lrDiameter, lrGearNumerator:= FB_MC2_AX5000_M_nMC_MotorParam1_lrGearNumerator, lrGearDenominator:= FB_MC2_AX5000_M_nMC_MotorParam1_lrGearDenominator);
	M_nMC_PID_PosCtrl(bExecute:= FB_MC2_AX5000_M_nMC_PID_PosCtrl_bExecute, rKv:= FB_MC2_AX5000_M_nMC_PID_PosCtrl_rKv);
	M_nMC_Torque(bExecute:= FB_MC2_AX5000_M_nMC_Torque_bExecute, lrTorque:= FB_MC2_AX5000_M_nMC_Torque_lrTorque);
	M_nMC_TouchProbe1(bEnable:= FB_MC2_AX5000_M_nMC_TouchProbe1_bEnable, lrPrellFilter_RisingEdge:= FB_MC2_AX5000_M_nMC_TouchProbe1_lrPrellFilter_RisingEdge);
	M_nMC_TouchProbe2(bEnable:= FB_MC2_AX5000_M_nMC_TouchProbe2_bEnable, lrPrellFilter_RisingEdge:= FB_MC2_AX5000_M_nMC_TouchProbe2_lrPrellFilter_RisingEdge, lrPrellFilter_FallingEdge:= FB_MC2_AX5000_M_nMC_TouchProbe2_lrPrellFilter_FallingEdge);
END_IF

//**********************************
// Call methods 
//**********************************
FB_MC2_AX5000_M_nMC_Power_fbStartDelay_TON(IN:= TRUE, PT:= T#200MS, Q=> , ET=> );
IF FB_MC2_AX5000_M_nMC_Power_fbStartDelay_TON.Q THEN
	IF _stAXIS_REF.NcToPlc.AxisID > 0 THEN
		FB_MC2_AX5000_M_nMC_Power_arr_nRet[1]:= SUPER^.M_nMC_Power(bEnable:= FB_MC2_AX5000_M_nMC_Power_bEnable, bE_Stop:= FB_MC2_AX5000_M_nMC_Power_bE_Stop, bE_StopDelay:= FB_MC2_AX5000_M_nMC_Power_bE_StopDelay, bEnable_Positive:= FB_MC2_AX5000_M_nMC_Power_bEnable_Positive, bEnable_Negative:= FB_MC2_AX5000_M_nMC_Power_bEnable_Negative);
		FB_MC2_AX5000_M_nMC_Power_arr_nRet[2]:= M_nMC_DriveData();				
	ELSE
		SUPER^.M_nMC_Power(bEnable:= FALSE, bE_Stop:= FB_MC2_AX5000_M_nMC_Power_bE_Stop, bE_StopDelay:= FB_MC2_AX5000_M_nMC_Power_bE_StopDelay, bEnable_Positive:= FB_MC2_AX5000_M_nMC_Power_bEnable_Positive, bEnable_Negative:= FB_MC2_AX5000_M_nMC_Power_bEnable_Negative);
		IF FB_MC2_AX5000_M_nMC_Power_bEnable THEN
			M_nMC_Power:= Tc3_HBI_System.cMAPPING_ERROR;
		END_IF
		RETURN;
	END_IF
END_IF


//**********************************
// Error handling
//**********************************
IF _stAXIS_REF.Status.Error THEN
	M_nError(_stAXIS_REF.Status.ErrorID);
	M_nMC_Power:= _nErrorID;
ELSE
	FOR _iIdx:= 1 TO UINT_TO_INT(SIZEOF(FB_MC2_AX5000_M_nMC_Power_arr_nRet) / SIZEOF(FB_MC2_AX5000_M_nMC_Power_arr_nRet[1])) DO
		IF FB_MC2_AX5000_M_nMC_Power_arr_nRet[_iIdx] > 5 AND FB_MC2_AX5000_M_nMC_Power_arr_nRet[_iIdx] <> 10 THEN
			M_nError(nErrorID:= FB_MC2_AX5000_M_nMC_Power_arr_nRet[_iIdx]);
			EXIT;
		END_IF
	END_FOR

	// Method return value
	IF _bError THEN
		M_nMC_Power:= _nErrorID;
	ELSE
		M_nMC_Power:= FB_MC2_AX5000_M_nMC_Power_arr_nRet[1];
	END_IF

END_IF
END_METHOD

//	The result of the method is an unsigned double integer
//	0 = idle 
//	1 = coupled
//	2 = starting
//	3 = running
//	4 = aborted
// 	5 = no hardware connected
// 	6 = Spare
//	7 = pointer or index error
//	8 = mapping error
//	9 = parameter error
//	10 = complete
//	Any other number = ErrorID
METHOD PUBLIC M_nMC_Torque : UDINT
VAR_INPUT
	bExecute: BOOL;
	lrTorque: LREAL; 		// Torque limit 0.0-100.0%	
END_VAR
// Local variable
FB_MC2_AX5000_M_nMC_Torque_bExecute:= bExecute;
FB_MC2_AX5000_M_nMC_Torque_lrTorque:= lrTorque;

//**********************************
// Reset 
//**********************************
IF _bReset THEN
	IF _bError THEN
		FB_MC2_AX5000_M_nMC_Torque_fbSoEWrite(Execute:= FALSE, Axis:= _stAXIS_REF); 
		FB_MC2_AX5000_M_nMC_Torque_fbExecute_R_TRIG(CLK:= FALSE);
		FB_MC2_AX5000_M_nMC_Torque_iState:= 000;
	END_IF
END_IF
// No hardware connected
IF NOT _bHardwareConnected THEN
	FB_MC2_AX5000_M_nMC_Torque_fbSoEWrite(Execute:= FALSE, Axis:= _stAXIS_REF); 
	FB_MC2_AX5000_M_nMC_Torque_fbExecute_R_TRIG(CLK:= FALSE);
	FB_MC2_AX5000_M_nMC_Torque_iState:= 000;
	IF FB_MC2_AX5000_M_nMC_Torque_bExecute THEN
		M_nMC_Torque:= Tc3_HBI_System.cNO_HARDWARE_CONNECTED;
	END_IF		
	RETURN;
END_IF

//**********************************
// Parameter check 
//**********************************
IF FB_MC2_AX5000_M_nMC_Torque_bExecute THEN
	IF FB_MC2_AX5000_M_nMC_Torque_lrTorque < 0.0 OR FB_MC2_AX5000_M_nMC_Torque_lrTorque > 100.0 THEN
		M_nMC_Torque:= Tc3_HBI_System.cPARAMETER_ERROR;
		
		FB_MC2_AX5000_M_nMC_Torque_fbSoEWrite(Execute:= FALSE, Axis:= _stAXIS_REF); 
		FB_MC2_AX5000_M_nMC_Torque_fbExecute_R_TRIG(CLK:= FALSE);
		FB_MC2_AX5000_M_nMC_Torque_iState:= 000;
		RETURN;
	END_IF
END_IF


//**********************************
// Wait for execute
//**********************************
IF _stAXIS_REF.NcToPlc.AxisID > 0 THEN
	FB_MC2_AX5000_M_nMC_Torque_fbExecute_R_TRIG(CLK:= FB_MC2_AX5000_M_nMC_Torque_bExecute);
	IF FB_MC2_AX5000_M_nMC_Torque_fbExecute_R_TRIG.Q THEN
		FB_MC2_AX5000_M_nMC_Torque_fbSoEWrite(Execute:= FALSE, Axis:= _stAXIS_REF); 
		FB_MC2_AX5000_M_nMC_Torque_iState:= 001;
	END_IF
ELSE
	FB_MC2_AX5000_M_nMC_Torque_fbExecute_R_TRIG(CLK:= FALSE);
	FB_MC2_AX5000_M_nMC_Torque_iState:= 000;
	IF FB_MC2_AX5000_M_nMC_Torque_bExecute THEN
		M_nMC_Torque:= Tc3_HBI_System.cMAPPING_ERROR;
	END_IF
	RETURN;
END_IF


//**********************************
// Main sequence
//**********************************
CASE FB_MC2_AX5000_M_nMC_Torque_iState OF

	000: 	// Do nothing
	
	001:	// Write torque limet	
			M_nMC_Torque:= Tc3_HBI_System.cRUNNING;
			FB_MC2_AX5000_M_nMC_Torque_iTorque:= LREAL_TO_INT(FB_MC2_AX5000_M_nMC_Torque_lrTorque * 10);
			FB_MC2_AX5000_M_nMC_Torque_fbSoEWrite(Execute:= FALSE, Axis:= _stAXIS_REF); 
			FB_MC2_AX5000_M_nMC_Torque_fbSoEWrite(
				NetId:= '', 
				Idn:= S_0_IDN + 92, 
				Element:= 16#40, 
				pSrcBuf:= ADR(FB_MC2_AX5000_M_nMC_Torque_iTorque), 
				BufLen:= SIZEOF(FB_MC2_AX5000_M_nMC_Torque_iTorque), 
				Execute:= TRUE, 
				Timeout:= Tc2_System.DEFAULT_ADS_TIMEOUT, 
				Password:= , 
				Axis:= _stAXIS_REF, 
				Busy=> , 
				Error=> , 
				AdsErrId=> , 
				SercosErrId=> );
	
			FB_MC2_AX5000_M_nMC_Torque_iState:= FB_MC2_AX5000_M_nMC_Torque_iState +1;

	002:	// Write torque limet
			M_nMC_Torque:= Tc3_HBI_System.cRUNNING;
			FB_MC2_AX5000_M_nMC_Torque_fbSoEWrite(Execute:= TRUE, Axis:= _stAXIS_REF); 
			
			// Error handling
			IF FB_MC2_AX5000_M_nMC_Torque_fbSoEWrite.Error THEN
				M_nError(FB_MC2_AX5000_M_nMC_Torque_fbSoEWrite.AdsErrId);
				M_nMC_Torque:= FB_MC2_AX5000_M_nMC_Torque_fbSoEWrite.AdsErrId;
			ELSE
				// Done
				IF NOT FB_MC2_AX5000_M_nMC_Torque_fbSoEWrite.Busy THEN
					FB_MC2_AX5000_M_nMC_Torque_fbSoEWrite(Execute:= FALSE, Axis:= _stAXIS_REF); 
					FB_MC2_AX5000_M_nMC_Torque_iState:= FB_MC2_AX5000_M_nMC_Torque_iState +1;
				END_IF	
			END_IF
		
	003:	// Done
			M_nMC_Torque:= Tc3_HBI_System.cCOMPLETE;
			IF NOT FB_MC2_AX5000_M_nMC_Torque_bExecute THEN
				FB_MC2_AX5000_M_nMC_Torque_iState:= 000;
			END_IF
		
ELSE
	FB_MC2_AX5000_M_nMC_Torque_iState:= 000;
END_CASE
END_METHOD

//	The result of the method is an unsigned double integer
//	0 = idle 
//	1 = coupled
//	2 = starting
//	3 = running
//	4 = aborted
// 	5 = no hardware connected
// 	6 = Spare
//	7 = pointer or index error
//	8 = mapping error
//	9 = parameter error
//	10 = complete
//	Any other number = ErrorID
METHOD PUBLIC M_nMC_TouchProbe1 : UDINT
VAR_INPUT
	bEnable: BOOL;
	lrPrellFilter_RisingEdge: LREAL;
END_VAR
// Local variable
FB_MC2_AX5000_M_nMC_TouchProbe1_bEnable:= bEnable;
FB_MC2_AX5000_M_nMC_TouchProbe1_lrPrellFilter_RisingEdge:= lrPrellFilter_RisingEdge;

//**********************************
// Reset 
//**********************************
IF _bReset THEN
	IF _bError THEN
		FB_MC2_AX5000_M_nMC_TouchProbe1_iState:= 000;
	END_IF
END_IF

// No hardware connected
IF NOT _bHardwareConnected THEN
	FB_MC2_AX5000_M_nMC_TouchProbe1_iState:= 000;
	IF FB_MC2_AX5000_M_nMC_TouchProbe1_bEnable THEN
		M_nMC_TouchProbe1:= Tc3_HBI_System.cNO_HARDWARE_CONNECTED;
	END_IF	
	RETURN;
END_IF

// Check for axis
IF _stAXIS_REF.NcToPlc.AxisID <= 0 THEN
	FB_MC2_AX5000_M_nMC_TouchProbe1_iState:= 000;
	IF FB_MC2_AX5000_M_nMC_TouchProbe1_bEnable THEN
		M_nMC_TouchProbe1:= Tc3_HBI_System.cNO_HARDWARE_CONNECTED;
	END_IF	
	RETURN;
END_IF

// Disable
FB_MC2_AX5000_M_nMC_TouchProbe1_fbDisable_R_TRIG(CLK:= NOT FB_MC2_AX5000_M_nMC_TouchProbe1_bEnable);
IF FB_MC2_AX5000_M_nMC_TouchProbe1_fbDisable_R_TRIG.Q THEN
	FB_MC2_AX5000_M_nMC_TouchProbe1_iState:= 000;
END_IF

// Enable
FB_MC2_AX5000_M_nMC_TouchProbe1_fbEnable_R_TRIG(CLK:= FB_MC2_AX5000_M_nMC_TouchProbe1_bEnable);
IF FB_MC2_AX5000_M_nMC_TouchProbe1_fbEnable_R_TRIG.Q THEN
	FB_MC2_AX5000_M_nMC_TouchProbe1_iState:= 000;
END_IF


//**********************************
// Main sequence
//**********************************
CASE FB_MC2_AX5000_M_nMC_TouchProbe1_iState OF

	000:	// Init TouchProbe
			M_nMC_TouchProbe1:= Tc3_HBI_System.cRUNNING;
			FB_MC2_AX5000_M_nMC_TouchProbe1_stTriggerInput.EncoderID:= _stAXIS_REF.NcToPlc.AxisId;
			FB_MC2_AX5000_M_nMC_TouchProbe1_stTriggerInput.Mode:= TC2_MC2.TOUCHPROBEMODE_SINGLE;
			FB_MC2_AX5000_M_nMC_TouchProbe1_stTriggerInput.TouchProbe:= TouchProbe1;
			FB_MC2_AX5000_M_nMC_TouchProbe1_stTriggerInput.Edge:= RisingEdge;	
			FB_MC2_AX5000_M_nMC_TouchProbe1_fbTouchProbe(Axis:= _stAXIS_REF, TriggerInput:= FB_MC2_AX5000_M_nMC_TouchProbe1_stTriggerInput, Execute:= FALSE, WindowOnly:= FALSE);
			FB_MC2_AX5000_M_nMC_TouchProbe1_fbAbortTrigger(Axis:= _stAXIS_REF,	TriggerInput:= FB_MC2_AX5000_M_nMC_TouchProbe1_stTriggerInput, Execute:= FALSE);
			FB_MC2_AX5000_M_nMC_TouchProbe1_lrRecordedPosition1_RisingEdge:= 0.0;
			FB_MC2_AX5000_M_nMC_TouchProbe1_lrLastLatchPosition:= 0.0;
			FB_MC2_AX5000_M_nMC_TouchProbe1_iState:= FB_MC2_AX5000_M_nMC_TouchProbe1_iState +1;

	001:	// MC_AbortTrigger
			M_nMC_TouchProbe1:= Tc3_HBI_System.cRUNNING;
			FB_MC2_AX5000_M_nMC_TouchProbe1_fbAbortTrigger(
				Axis:= _stAXIS_REF, 
				TriggerInput:= FB_MC2_AX5000_M_nMC_TouchProbe1_stTriggerInput, 
				Execute:= TRUE, 
				Done=> , 
				Busy=> , 
				Error=> , 
				ErrorID=> );		

			// Error handling
			IF FB_MC2_AX5000_M_nMC_TouchProbe1_fbAbortTrigger.Error THEN
				IF 	FB_MC2_AX5000_M_nMC_TouchProbe1_fbAbortTrigger.ErrorID = 17460 THEN
					IF FB_MC2_AX5000_M_nMC_TouchProbe1_bEnable THEN
						M_nError(nErrorID:= FB_MC2_AX5000_M_nMC_TouchProbe1_fbAbortTrigger.ErrorID);
						M_nMC_TouchProbe1:= FB_MC2_AX5000_M_nMC_TouchProbe1_fbAbortTrigger.ErrorID;
					ELSE
						FB_MC2_AX5000_M_nMC_TouchProbe1_fbAbortTrigger(Axis:= _stAXIS_REF, TriggerInput:= FB_MC2_AX5000_M_nMC_TouchProbe1_stTriggerInput, Execute:= FALSE);
						FB_MC2_AX5000_M_nMC_TouchProbe1_iState:= FB_MC2_AX5000_M_nMC_TouchProbe1_iState +1;
					END_IF
				ELSE
					M_nError(nErrorID:= FB_MC2_AX5000_M_nMC_TouchProbe1_fbAbortTrigger.ErrorID);
					M_nMC_TouchProbe1:= FB_MC2_AX5000_M_nMC_TouchProbe1_fbAbortTrigger.ErrorID;
				END_IF
			ELSE
				// Done
				IF FB_MC2_AX5000_M_nMC_TouchProbe1_fbAbortTrigger.Done THEN
					FB_MC2_AX5000_M_nMC_TouchProbe1_fbAbortTrigger(Axis:= _stAXIS_REF, TriggerInput:= FB_MC2_AX5000_M_nMC_TouchProbe1_stTriggerInput, Execute:= FALSE);
					FB_MC2_AX5000_M_nMC_TouchProbe1_iState:= FB_MC2_AX5000_M_nMC_TouchProbe1_iState +1;
				END_IF	
			END_IF
	
	002:	// Wait for bEnable
			IF FB_MC2_AX5000_M_nMC_TouchProbe1_bEnable THEN
				FB_MC2_AX5000_M_nMC_TouchProbe1_iState:= 010;
			END_IF
	
	010:	// TouchProbe rising edge	
			M_nMC_TouchProbe1:= Tc3_HBI_System.cRUNNING;
			IF FB_MC2_AX5000_M_nMC_TouchProbe1_bEnable THEN
				
				FB_MC2_AX5000_M_nMC_TouchProbe1_fbTouchProbe(Axis:= _stAXIS_REF, TriggerInput:= FB_MC2_AX5000_M_nMC_TouchProbe2_stTriggerInput, Execute:= TRUE, WindowOnly:= FALSE);
				
				// Error handling
				IF FB_MC2_AX5000_M_nMC_TouchProbe1_fbTouchProbe.Error THEN
					IF 	FB_MC2_AX5000_M_nMC_TouchProbe1_fbTouchProbe.ErrorID = 19212 THEN
						FB_MC2_AX5000_M_nMC_TouchProbe1_fbTouchProbe(Axis:= _stAXIS_REF, TriggerInput:= FB_MC2_AX5000_M_nMC_TouchProbe1_stTriggerInput, Execute:= FALSE, WindowOnly:= FALSE);
					ELSE
						M_nError(nErrorID:= FB_MC2_AX5000_M_nMC_TouchProbe1_fbTouchProbe.ErrorID);
						M_nMC_TouchProbe1:= FB_MC2_AX5000_M_nMC_TouchProbe1_fbTouchProbe.ErrorID;
					END_IF
				ELSE
					// Aborted	
					IF FB_MC2_AX5000_M_nMC_TouchProbe1_fbTouchProbe.CommandAborted THEN
						FB_MC2_AX5000_M_nMC_TouchProbe1_iState:= 000;
					ELSE
						// Done
						IF FB_MC2_AX5000_M_nMC_TouchProbe1_fbTouchProbe.Done THEN

							// Prellfilter 
							IF ABS(_stAXIS_REF.NcToPlc.ActPos - FB_MC2_AX5000_M_nMC_TouchProbe1_lrLastLatchPosition) >= FB_MC2_AX5000_M_nMC_TouchProbe1_lrPrellFilter_RisingEdge THEN
								FB_MC2_AX5000_M_nMC_TouchProbe1_lrRecordedPosition1_RisingEdge:= FB_MC2_AX5000_M_nMC_TouchProbe1_fbTouchProbe.RecordedPosition;
								FB_MC2_AX5000_M_nMC_TouchProbe1_lrLastLatchPosition:= FB_MC2_AX5000_M_nMC_TouchProbe1_fbTouchProbe.RecordedPosition;
								M_nMC_TouchProbe1:= Tc3_HBI_System.cCOMPLETE;				
							END_IF
								
							FB_MC2_AX5000_M_nMC_TouchProbe1_fbTouchProbe(Axis:= _stAXIS_REF, TriggerInput:= FB_MC2_AX5000_M_nMC_TouchProbe1_stTriggerInput, Execute:= FALSE, WindowOnly:= FALSE);
						END_IF
					END_IF	
				END_IF			
				
			ELSE
				FB_MC2_AX5000_M_nMC_TouchProbe1_iState:= 000;
			END_IF
		
ELSE
	FB_MC2_AX5000_M_nMC_TouchProbe1_iState:= 0;
END_CASE
END_METHOD

//	The result of the method is an unsigned double integer
//	0 = idle 
//	1 = coupled
//	2 = starting
//	3 = running
//	4 = aborted
// 	5 = no hardware connected
// 	6 = Spare
//	7 = pointer or index error
//	8 = mapping error
//	9 = parameter error
//	10 = complete
//	Any other number = ErrorID
METHOD PUBLIC M_nMC_TouchProbe2 : UDINT
VAR_INPUT
	bEnable: BOOL;
	lrPrellFilter_RisingEdge: LREAL;
	lrPrellFilter_FallingEdge: LREAL;
END_VAR
// Local variable
FB_MC2_AX5000_M_nMC_TouchProbe2_bEnable:= bEnable;
FB_MC2_AX5000_M_nMC_TouchProbe2_lrPrellFilter_RisingEdge:= lrPrellFilter_RisingEdge;
FB_MC2_AX5000_M_nMC_TouchProbe2_lrPrellFilter_FallingEdge:= lrPrellFilter_FallingEdge;

//**********************************
// Reset 
//**********************************
IF _bReset THEN
	IF _bError THEN
		FB_MC2_AX5000_M_nMC_TouchProbe2_iState:= 000;
	END_IF
END_IF

// No hardware connected
IF NOT _bHardwareConnected THEN
	FB_MC2_AX5000_M_nMC_TouchProbe2_iState:= 000;
	IF FB_MC2_AX5000_M_nMC_TouchProbe2_bEnable THEN
		M_nMC_TouchProbe2:= Tc3_HBI_System.cNO_HARDWARE_CONNECTED;
	END_IF	
	RETURN;	
END_IF

// Check for axis
IF _stAXIS_REF.NcToPlc.AxisID <= 0 THEN
	FB_MC2_AX5000_M_nMC_TouchProbe2_iState:= 000;
	IF FB_MC2_AX5000_M_nMC_TouchProbe2_bEnable THEN
		M_nMC_TouchProbe2:= Tc3_HBI_System.cNO_HARDWARE_CONNECTED;
	END_IF	
	RETURN;	
END_IF

// Disable
FB_MC2_AX5000_M_nMC_TouchProbe2_fbDisable_R_TRIG(CLK:= NOT FB_MC2_AX5000_M_nMC_TouchProbe2_bEnable);
IF FB_MC2_AX5000_M_nMC_TouchProbe2_fbDisable_R_TRIG.Q THEN
	FB_MC2_AX5000_M_nMC_TouchProbe2_iState:= 000;
END_IF

// Enable
FB_MC2_AX5000_M_nMC_TouchProbe2_fbEnable_R_TRIG(CLK:= FB_MC2_AX5000_M_nMC_TouchProbe2_bEnable);
IF FB_MC2_AX5000_M_nMC_TouchProbe2_fbEnable_R_TRIG.Q THEN
	FB_MC2_AX5000_M_nMC_TouchProbe2_iState:= 000;
END_IF


//**********************************
// Main sequence
//**********************************
CASE FB_MC2_AX5000_M_nMC_TouchProbe2_iState OF

	000:	// Init TouchProbe
			M_nMC_TouchProbe2:= Tc3_HBI_System.cRUNNING;
			FB_MC2_AX5000_M_nMC_TouchProbe2_stTriggerInput.EncoderID:= _stAXIS_REF.NcToPlc.AxisId;
			FB_MC2_AX5000_M_nMC_TouchProbe2_stTriggerInput.Mode:= TC2_MC2.TOUCHPROBEMODE_SINGLE;
			FB_MC2_AX5000_M_nMC_TouchProbe2_fbTouchProbe(Axis:= _stAXIS_REF, TriggerInput:= FB_MC2_AX5000_M_nMC_TouchProbe2_stTriggerInput, Execute:= FALSE, WindowOnly:= FALSE);
			FB_MC2_AX5000_M_nMC_TouchProbe2_fbAbortTrigger(Axis:= _stAXIS_REF,	TriggerInput:= FB_MC2_AX5000_M_nMC_TouchProbe2_stTriggerInput, Execute:= FALSE);
			FB_MC2_AX5000_M_nMC_TouchProbe2_lrRecordedPosition2_RisingEdge:= 0.0;
			FB_MC2_AX5000_M_nMC_TouchProbe2_lrRecordedPosition2_FallingEdge:= 0.0;
			FB_MC2_AX5000_M_nMC_TouchProbe2_iState:= FB_MC2_AX5000_M_nMC_TouchProbe2_iState +1;

	001:	// MC_AbortTrigger RisingEdge
			M_nMC_TouchProbe2:= Tc3_HBI_System.cRUNNING;
			FB_MC2_AX5000_M_nMC_TouchProbe2_stTriggerInput.Edge:= Tc2_MC2.RisingEdge;				
			FB_MC2_AX5000_M_nMC_TouchProbe2_fbAbortTrigger(
				Axis:= _stAXIS_REF, 
				TriggerInput:= FB_MC2_AX5000_M_nMC_TouchProbe2_stTriggerInput, 
				Execute:= TRUE, 
				Done=> , 
				Busy=> , 
				Error=> , 
				ErrorID=> );		
				
			// Error handling
			IF FB_MC2_AX5000_M_nMC_TouchProbe2_fbAbortTrigger.Error THEN
				IF 	FB_MC2_AX5000_M_nMC_TouchProbe2_fbAbortTrigger.ErrorID = 17460 THEN
					IF FB_MC2_AX5000_M_nMC_TouchProbe2_bEnable THEN
						M_nError(nErrorID:= FB_MC2_AX5000_M_nMC_TouchProbe2_fbAbortTrigger.ErrorID);
						M_nMC_TouchProbe2:= FB_MC2_AX5000_M_nMC_TouchProbe2_fbAbortTrigger.ErrorID;
					ELSE
						FB_MC2_AX5000_M_nMC_TouchProbe2_fbAbortTrigger(Axis:= _stAXIS_REF, TriggerInput:= FB_MC2_AX5000_M_nMC_TouchProbe2_stTriggerInput, Execute:= FALSE);
						FB_MC2_AX5000_M_nMC_TouchProbe2_iState:= FB_MC2_AX5000_M_nMC_TouchProbe2_iState +1;
					END_IF
				ELSE
					M_nError(nErrorID:= FB_MC2_AX5000_M_nMC_TouchProbe2_fbAbortTrigger.ErrorID);
					M_nMC_TouchProbe2:= FB_MC2_AX5000_M_nMC_TouchProbe2_fbAbortTrigger.ErrorID;
				END_IF
			ELSE
				IF FB_MC2_AX5000_M_nMC_TouchProbe2_fbAbortTrigger.Done THEN
					FB_MC2_AX5000_M_nMC_TouchProbe2_fbAbortTrigger(Axis:= _stAXIS_REF, TriggerInput:= FB_MC2_AX5000_M_nMC_TouchProbe2_stTriggerInput, Execute:= FALSE);
					FB_MC2_AX5000_M_nMC_TouchProbe2_iState:= FB_MC2_AX5000_M_nMC_TouchProbe2_iState +1;
				END_IF	
			END_IF	
				
	002:	// MC_AbortTrigger FallingEdge
			M_nMC_TouchProbe2:= Tc3_HBI_System.cRUNNING;
			FB_MC2_AX5000_M_nMC_TouchProbe2_stTriggerInput.Edge:= Tc2_MC2.FallingEdge;			
			FB_MC2_AX5000_M_nMC_TouchProbe2_fbAbortTrigger(
				Axis:= _stAXIS_REF, 
				TriggerInput:= FB_MC2_AX5000_M_nMC_TouchProbe2_stTriggerInput, 
				Execute:= TRUE, 
				Done=> , 
				Busy=> , 
				Error=> , 
				ErrorID=> );		
				
			// Error handling
			IF FB_MC2_AX5000_M_nMC_TouchProbe2_fbAbortTrigger.Error THEN
				IF 	FB_MC2_AX5000_M_nMC_TouchProbe2_fbAbortTrigger.ErrorID = 17460 THEN
					IF FB_MC2_AX5000_M_nMC_TouchProbe2_bEnable THEN
						M_nError(nErrorID:= FB_MC2_AX5000_M_nMC_TouchProbe2_fbAbortTrigger.ErrorID);
						M_nMC_TouchProbe2:= FB_MC2_AX5000_M_nMC_TouchProbe2_fbAbortTrigger.ErrorID;
					ELSE
						FB_MC2_AX5000_M_nMC_TouchProbe2_fbAbortTrigger(Axis:= _stAXIS_REF, TriggerInput:= FB_MC2_AX5000_M_nMC_TouchProbe2_stTriggerInput, Execute:= FALSE);
						FB_MC2_AX5000_M_nMC_TouchProbe2_iState:= FB_MC2_AX5000_M_nMC_TouchProbe2_iState +1;
					END_IF
				ELSE
					M_nError(nErrorID:= FB_MC2_AX5000_M_nMC_TouchProbe2_fbAbortTrigger.ErrorID);
					M_nMC_TouchProbe2:= FB_MC2_AX5000_M_nMC_TouchProbe2_fbAbortTrigger.ErrorID;
				END_IF
			ELSE
				IF FB_MC2_AX5000_M_nMC_TouchProbe2_fbAbortTrigger.Done THEN
					FB_MC2_AX5000_M_nMC_TouchProbe2_fbAbortTrigger(Axis:= _stAXIS_REF, TriggerInput:= FB_MC2_AX5000_M_nMC_TouchProbe2_stTriggerInput, Execute:= FALSE);
					FB_MC2_AX5000_M_nMC_TouchProbe2_iState:= FB_MC2_AX5000_M_nMC_TouchProbe2_iState +1;
				END_IF	
			END_IF	
			
	003:	// Wait for bEnable
			FB_MC2_AX5000_M_nMC_TouchProbe2_stTriggerInput.Edge:= Tc2_MC2.RisingEdge;				
			IF FB_MC2_AX5000_M_nMC_TouchProbe2_bEnable THEN
				FB_MC2_AX5000_M_nMC_TouchProbe2_iState:= 010;
			END_IF

	010:	// Touch probe handling
			M_nMC_TouchProbe2:= Tc3_HBI_System.cRUNNING;
			IF FB_MC2_AX5000_M_nMC_TouchProbe2_bEnable THEN

				FB_MC2_AX5000_M_nMC_TouchProbe2_fbTouchProbe(Axis:= _stAXIS_REF, TriggerInput:= FB_MC2_AX5000_M_nMC_TouchProbe2_stTriggerInput, Execute:= TRUE, WindowOnly:= FALSE);
			
				// Error handling
				IF FB_MC2_AX5000_M_nMC_TouchProbe2_fbTouchProbe.Error THEN
					IF 	FB_MC2_AX5000_M_nMC_TouchProbe2_fbTouchProbe.ErrorID = 19212 THEN
						FB_MC2_AX5000_M_nMC_TouchProbe2_fbTouchProbe(Axis:= _stAXIS_REF, TriggerInput:= FB_MC2_AX5000_M_nMC_TouchProbe2_stTriggerInput, Execute:= FALSE, WindowOnly:= FALSE);
					ELSE
						M_nError(nErrorID:= FB_MC2_AX5000_M_nMC_TouchProbe2_fbTouchProbe.ErrorID);
						M_nMC_TouchProbe2:= FB_MC2_AX5000_M_nMC_TouchProbe2_fbTouchProbe.ErrorID;
					END_IF
				ELSE
					// Aborted	
					IF FB_MC2_AX5000_M_nMC_TouchProbe2_fbTouchProbe.CommandAborted THEN
						FB_MC2_AX5000_M_nMC_TouchProbe2_iState:= 000;
					ELSE
						// Done
						IF FB_MC2_AX5000_M_nMC_TouchProbe2_fbTouchProbe.Done THEN
							IF FB_MC2_AX5000_M_nMC_TouchProbe2_stTriggerInput.Edge = Tc2_MC2.RisingEdge THEN

								// Prellfilter 
								IF ABS(_stAXIS_REF.NcToPlc.ActPos - FB_MC2_AX5000_M_nMC_TouchProbe2_lrLastLatchPosition) >= FB_MC2_AX5000_M_nMC_TouchProbe2_lrPrellFilter_FallingEdge THEN
									IF NOT FB_MC2_AX5000_M_nMC_TouchProbe2_bRisingEdgeDone THEN
										FB_MC2_AX5000_M_nMC_TouchProbe2_lrLastLatchPosition:= FB_MC2_AX5000_M_nMC_TouchProbe2_fbTouchProbe.RecordedPosition;
									END_IF	
									FB_MC2_AX5000_M_nMC_TouchProbe2_bRisingEdgeDone:= TRUE;									
								END_IF
								
								FB_MC2_AX5000_M_nMC_TouchProbe2_stTriggerInput.Edge:= Tc2_MC2.FallingEdge;
							ELSE

								// Prellfilter 
								IF ABS(_stAXIS_REF.NcToPlc.ActPos - FB_MC2_AX5000_M_nMC_TouchProbe2_lrLastLatchPosition) >= FB_MC2_AX5000_M_nMC_TouchProbe2_lrPrellFilter_RisingEdge THEN
									IF FB_MC2_AX5000_M_nMC_TouchProbe2_bRisingEdgeDone THEN
										FB_MC2_AX5000_M_nMC_TouchProbe2_lrRecordedPosition2_RisingEdge:= FB_MC2_AX5000_M_nMC_TouchProbe2_lrLastLatchPosition;
										FB_MC2_AX5000_M_nMC_TouchProbe2_lrRecordedPosition2_FallingEdge:= FB_MC2_AX5000_M_nMC_TouchProbe2_fbTouchProbe.RecordedPosition;
										FB_MC2_AX5000_M_nMC_TouchProbe2_lrLastLatchPosition:= FB_MC2_AX5000_M_nMC_TouchProbe2_fbTouchProbe.RecordedPosition;
										FB_MC2_AX5000_M_nMC_TouchProbe2_bRisingEdgeDone:= FALSE;
										M_nMC_TouchProbe2:= Tc3_HBI_System.cCOMPLETE;				
									END_IF	
								END_IF
								
